LIN {X 0,Y 523.916,Z 118.035,A -85,B 0,C 180,E1 -4641.08,E2 -4641.08} C_VEL
LIN {X 0,Y 523.924,Z 118.033,A -85,B 0,C 180,E1 -4643.827,E2 -4643.827} C_VEL
LIN {X 0,Y 523.941,Z 118.03,A -85,B 0,C 180,E1 -4646.635,E2 -4646.635} C_VEL
LIN {X 0,Y 523.955,Z 118.032,A -85,B 0,C 180,E1 -4649.356,E2 -4649.356} C_VEL
LIN {X 0,Y 523.976,Z 118.024,A -85,B 0,C 180,E1 -4652.281,E2 -4652.281} C_VEL
LIN {X 0,Y 523.951,Z 118.031,A -85,B 0,C 180,E1 -4654.581,E2 -4654.581} C_VEL
LIN {X 0,Y 523.91,Z 118.037,A -85,B 0,C 180,E1 -4657.106,E2 -4657.106} C_VEL
LIN {X 0,Y 523.978,Z 118.024,A -85,B 0,C 180,E1 -4659.866,E2 -4659.866} C_VEL
LIN {X 0,Y 523.966,Z 118.031,A -85,B 0,C 180,E1 -4662.837,E2 -4662.837} C_VEL
LIN {X 0,Y 523.976,Z 118.025,A -85,B 0,C 180,E1 -4665.236,E2 -4665.236} C_VEL
LIN {X 0,Y 524.014,Z 118.028,A -85,B 0,C 180,E1 -4668.394,E2 -4668.394} C_VEL
LIN {X 0,Y 524.002,Z 118.021,A -85,B 0,C 180,E1 -4671.516,E2 -4671.516} C_VEL
LIN {X 0,Y 524.081,Z 118.014,A -85,B 0,C 180,E1 -4674.614,E2 -4674.614} C_VEL
LIN {X 0,Y 524.112,Z 118.011,A -85,B 0,C 180,E1 -4677.694,E2 -4677.694} C_VEL
LIN {X 0,Y 524.122,Z 118.006,A -85,B 0,C 180,E1 -4680.768,E2 -4680.768} C_VEL
LIN {X 0,Y 524.07,Z 118.013,A -85,B 0,C 180,E1 -4683.075,E2 -4683.075} C_VEL
LIN {X 0,Y 524.045,Z 118.018,A -85,B 0,C 180,E1 -4686.159,E2 -4686.159} C_VEL
LIN {X 0,Y 523.996,Z 118.025,A -85,B 0,C 180,E1 -4689.262,E2 -4689.262} C_VEL
LIN {X 0,Y 524.001,Z 118.026,A -85,B 0,C 180,E1 -4691.739,E2 -4691.739} C_VEL
LIN {X 0,Y 523.992,Z 118.026,A -85,B 0,C 180,E1 -4695.052,E2 -4695.052} C_VEL
LIN {X 0,Y 523.963,Z 118.026,A -85,B 0,C 180,E1 -4697.969,E2 -4697.969} C_VEL
LIN {X 0,Y 523.971,Z 118.025,A -85,B 0,C 180,E1 -4700.41,E2 -4700.41} C_VEL
LIN {X 0,Y 523.909,Z 118.038,A -85,B 0,C 180,E1 -4702.894,E2 -4702.894} C_VEL
LIN {X 0,Y 523.95,Z 118.03,A -85,B 0,C 180,E1 -4705.419,E2 -4705.419} C_VEL
LIN {X 0,Y 523.966,Z 118.025,A -85,B 0,C 180,E1 -4707.999,E2 -4707.999} C_VEL
LIN {X 0,Y 523.943,Z 118.036,A -85,B 0,C 180,E1 -4710.855,E2 -4710.855} C_VEL
LIN {X 0,Y 523.959,Z 118.026,A -85,B 0,C 180,E1 -4713.735,E2 -4713.735} C_VEL
LIN {X 0,Y 523.918,Z 118.037,A -85,B 0,C 180,E1 -4716.404,E2 -4716.404} C_VEL
LIN {X 0,Y 523.918,Z 118.032,A -85,B 0,C 180,E1 -4719.085,E2 -4719.085} C_VEL
LIN {X 0,Y 523.952,Z 118.032,A -85,B 0,C 180,E1 -4722.119,E2 -4722.119} C_VEL
LIN {X 0,Y 523.942,Z 118.028,A -85,B 0,C 180,E1 -4725.31,E2 -4725.31} C_VEL
LIN {X 0,Y 523.956,Z 118.028,A -85,B 0,C 180,E1 -4728.69,E2 -4728.69} C_VEL
LIN {X 0,Y 523.915,Z 118.031,A -85,B 0,C 180,E1 -4731.081,E2 -4731.081} C_VEL
LIN {X 0,Y 523.922,Z 118.038,A -85,B 0,C 180,E1 -4733.827,E2 -4733.827} C_VEL
LIN {X 0,Y 523.913,Z 118.032,A -85,B 0,C 180,E1 -4736.634,E2 -4736.634} C_VEL
LIN {X 0,Y 523.955,Z 118.03,A -85,B 0,C 180,E1 -4739.356,E2 -4739.356} C_VEL
LIN {X 0,Y 523.976,Z 118.025,A -85,B 0,C 180,E1 -4742.282,E2 -4742.282} C_VEL
LIN {X 0,Y 523.951,Z 118.028,A -85,B 0,C 180,E1 -4744.582,E2 -4744.582} C_VEL
LIN {X 0,Y 523.909,Z 118.018,A -85,B 0,C 180,E1 -4747.107,E2 -4747.107} C_VEL
LIN {X 0,Y 523.971,Z 118.238,A -85,B 0,C 180,E1 -4748.097,E2 -4748.097} C_VEL
LIN {X 0,Y 524.691,Z 123.717,A -85,B 0,C 180,E1 -4749.21,E2 -4749.21} C_VEL
LIN {X 0,Y 524.349,Z 138.793,A -85,B 0,C 180,E1 -4752.107,E2 -4752.107} C_VEL
LIN {X 0,Y 524.033,Z 153.682,A -85,B 0,C 180,E1 -4754.932,E2 -4754.932} C_VEL
LIN {X 0,Y 523.832,Z 170.237,A -85,B 0,C 180,E1 -4758.019,E2 -4758.019} C_VEL
LIN {X 0,Y 523.848,Z 170.802,A -85,B 0,C 180,E1 -4758.075,E2 -4758.075} C_VEL
LIN {X 0,Y 524.951,Z 180.485,A -85,B 0,C 180,E1 -4758.254,E2 -4758.254} C_VEL
LIN {X 0,Y 524.795,Z 246.49,A -85,B 0,C 180,E1 -4759.17,E2 -4759.17} C_VEL
LIN {X 0,Y 524.624,Z 255.76,A -85,B 0,C 180,E1 -4759.386,E2 -4759.386} C_VEL
LIN {X 0,Y 524.521,Z 264.237,A -85,B 0,C 180,E1 -4759.676,E2 -4759.676} C_VEL
LIN {X 0,Y 524.401,Z 272.75,A -85,B 0,C 180,E1 -4760.064,E2 -4760.064} C_VEL
LIN {X 0,Y 524.221,Z 281.094,A -85,B 0,C 180,E1 -4760.548,E2 -4760.548} C_VEL
LIN {X 0,Y 524.065,Z 289.144,A -85,B 0,C 180,E1 -4761.129,E2 -4761.129} C_VEL
LIN {X 0,Y 523.853,Z 297.832,A -85,B 0,C 180,E1 -4761.902,E2 -4761.902} C_VEL
LIN {X 0,Y 523.702,Z 306.356,A -85,B 0,C 180,E1 -4762.869,E2 -4762.869} C_VEL
LIN {X 0,Y 523.612,Z 313.045,A -85,B 0,C 180,E1 -4763.836,E2 -4763.836} C_VEL
LIN {X 0,Y 523.484,Z 317.435,A -85,B 0,C 180,E1 -4764.608,E2 -4764.608} C_VEL
LIN {X 0,Y 523.465,Z 322.611,A -85,B 0,C 180,E1 -4765.765,E2 -4765.765} C_VEL
LIN {X 0,Y 523.407,Z 325.256,A -85,B 0,C 180,E1 -4766.536,E2 -4766.536} C_VEL
LIN {X 0,Y 523.336,Z 328.158,A -85,B 0,C 180,E1 -4767.691,E2 -4767.691} C_VEL
LIN {X 0,Y 523.273,Z 329.409,A -85,B 0,C 180,E1 -4768.461,E2 -4768.461} C_VEL
LIN {X 0,Y 523.248,Z 330.188,A -85,B 0,C 180,E1 -4769.231,E2 -4769.231} C_VEL
LIN {X 0,Y 523.247,Z 330.484,A -85,B 0,C 180,E1 -4770,E2 -4770} C_VEL
LIN {X 0,Y 523.248,Z 330.188,A -85,B 0,C 180,E1 -4770.77,E2 -4770.77} C_VEL
LIN {X 0,Y 523.273,Z 329.408,A -85,B 0,C 180,E1 -4771.539,E2 -4771.539} C_VEL
LIN {X 0,Y 523.336,Z 328.156,A -85,B 0,C 180,E1 -4772.309,E2 -4772.309} C_VEL
LIN {X 0,Y 523.407,Z 325.254,A -85,B 0,C 180,E1 -4773.464,E2 -4773.464} C_VEL
LIN {X 0,Y 523.465,Z 322.609,A -85,B 0,C 180,E1 -4774.235,E2 -4774.235} C_VEL
LIN {X 0,Y 523.484,Z 317.43,A -85,B 0,C 180,E1 -4775.393,E2 -4775.393} C_VEL
LIN {X 0,Y 523.599,Z 311.458,A -85,B 0,C 180,E1 -4776.424,E2 -4776.424} C_VEL
LIN {X 0,Y 523.697,Z 304.846,A -85,B 0,C 180,E1 -4777.325,E2 -4777.325} C_VEL
LIN {X 0,Y 523.897,Z 296.813,A -85,B 0,C 180,E1 -4778.195,E2 -4778.195} C_VEL
LIN {X 0,Y 524.065,Z 289.143,A -85,B 0,C 180,E1 -4778.872,E2 -4778.872} C_VEL
LIN {X 0,Y 524.24,Z 281.089,A -85,B 0,C 180,E1 -4779.452,E2 -4779.452} C_VEL
LIN {X 0,Y 524.394,Z 272.745,A -85,B 0,C 180,E1 -4779.936,E2 -4779.936} C_VEL
LIN {X 0,Y 524.546,Z 264.232,A -85,B 0,C 180,E1 -4780.323,E2 -4780.323} C_VEL
LIN {X 0,Y 524.635,Z 254.085,A -85,B 0,C 180,E1 -4780.663,E2 -4780.663} C_VEL
LIN {X 0,Y 524.826,Z 242.383,A -85,B 0,C 180,E1 -4780.903,E2 -4780.903} C_VEL
LIN {X 0,Y 524.778,Z 178.186,A -85,B 0,C 180,E1 -4781.782,E2 -4781.782} C_VEL
LIN {X 0,Y 523.851,Z 170.702,A -85,B 0,C 180,E1 -4781.93,E2 -4781.93} C_VEL
LIN {X 0,Y 523.841,Z 164.752,A -85,B 0,C 180,E1 -4782.987,E2 -4782.987} C_VEL
LIN {X 0,Y 524.091,Z 151.089,A -85,B 0,C 180,E1 -4785.557,E2 -4785.557} C_VEL
LIN {X 0,Y 524.457,Z 134.255,A -85,B 0,C 180,E1 -4788.761,E2 -4788.761} C_VEL
LIN {X 0,Y 524.69,Z 122.657,A -85,B 0,C 180,E1 -4790.996,E2 -4790.996} C_VEL
LIN {X 0,Y 523.958,Z 118.102,A -85,B 0,C 180,E1 -4791.956,E2 -4791.956} C_VEL
LIN {X 0,Y 523.929,Z 118.024,A -85,B 0,C 180,E1 -4794.572,E2 -4794.572} C_VEL
LIN {X 0,Y 523.951,Z 118.028,A -85,B 0,C 180,E1 -4797.133,E2 -4797.133} C_VEL
LIN {X 0,Y 523.943,Z 118.03,A -85,B 0,C 180,E1 -4799.756,E2 -4799.756} C_VEL
LIN {X 0,Y 523.934,Z 118.035,A -85,B 0,C 180,E1 -4802.45,E2 -4802.45} C_VEL
LIN {X 0,Y 523.921,Z 118.031,A -85,B 0,C 180,E1 -4805.227,E2 -4805.227} C_VEL
LIN {X 0,Y 523.916,Z 118.039,A -85,B 0,C 180,E1 -4808.102,E2 -4808.102} C_VEL
LIN {X 0,Y 523.939,Z 118.029,A -85,B 0,C 180,E1 -4811.092,E2 -4811.092} C_VEL
LIN {X 0,Y 523.931,Z 118.032,A -85,B 0,C 180,E1 -4814.229,E2 -4814.229} C_VEL
LIN {X 0,Y 523.917,Z 118.031,A -85,B 0,C 180,E1 -4816.833,E2 -4816.833} C_VEL
LIN {X 0,Y 523.941,Z 118.029,A -85,B 0,C 180,E1 -4818.908,E2 -4818.908} C_VEL
LIN {X 0,Y 523.917,Z 118.035,A -85,B 0,C 180,E1 -4821.898,E2 -4821.898} C_VEL
LIN {X 0,Y 523.936,Z 118.031,A -85,B 0,C 180,E1 -4824.91,E2 -4824.91} C_VEL
LIN {X 0,Y 523.936,Z 118.032,A -85,B 0,C 180,E1 -4827.68,E2 -4827.68} C_VEL
LIN {X 0,Y 523.955,Z 118.029,A -85,B 0,C 180,E1 -4830.677,E2 -4830.677} C_VEL
LIN {X 0,Y 523.974,Z 118.025,A -85,B 0,C 180,E1 -4833.729,E2 -4833.729} C_VEL
LIN {X 0,Y 523.926,Z 118.031,A -85,B 0,C 180,E1 -4836.27,E2 -4836.27} C_VEL
LIN {X 0,Y 523.948,Z 118.035,A -85,B 0,C 180,E1 -4838.767,E2 -4838.767} C_VEL
LIN {X 0,Y 523.953,Z 118.03,A -85,B 0,C 180,E1 -4841.221,E2 -4841.221} C_VEL
LIN {X 0,Y 523.938,Z 118.029,A -85,B 0,C 180,E1 -4843.639,E2 -4843.639} C_VEL
LIN {X 0,Y 523.941,Z 118.03,A -85,B 0,C 180,E1 -4846.028,E2 -4846.028} C_VEL
LIN {X 0,Y 524.014,Z 118.026,A -85,B 0,C 180,E1 -4848.394,E2 -4848.394} C_VEL
LIN {X 0,Y 524.005,Z 118.02,A -85,B 0,C 180,E1 -4851.516,E2 -4851.516} C_VEL
LIN {X 0,Y 524.082,Z 118.015,A -85,B 0,C 180,E1 -4854.614,E2 -4854.614} C_VEL
LIN {X 0,Y 524.112,Z 118.01,A -85,B 0,C 180,E1 -4857.695,E2 -4857.695} C_VEL
LIN {X 0,Y 524.125,Z 118.006,A -85,B 0,C 180,E1 -4860.768,E2 -4860.768} C_VEL
LIN {X 0,Y 524.071,Z 118.012,A -85,B 0,C 180,E1 -4863.075,E2 -4863.075} C_VEL
LIN {X 0,Y 524.047,Z 118.019,A -85,B 0,C 180,E1 -4866.159,E2 -4866.159} C_VEL
LIN {X 0,Y 523.998,Z 118.024,A -85,B 0,C 180,E1 -4869.262,E2 -4869.262} C_VEL
LIN {X 0,Y 524.027,Z 118.025,A -85,B 0,C 180,E1 -4871.751,E2 -4871.751} C_VEL
LIN {X 0,Y 523.995,Z 118.024,A -85,B 0,C 180,E1 -4875.052,E2 -4875.052} C_VEL
LIN {X 0,Y 523.965,Z 118.027,A -85,B 0,C 180,E1 -4877.969,E2 -4877.969} C_VEL
LIN {X 0,Y 523.974,Z 118.024,A -85,B 0,C 180,E1 -4880.41,E2 -4880.41} C_VEL
LIN {X 0,Y 523.912,Z 118.036,A -85,B 0,C 180,E1 -4882.894,E2 -4882.894} C_VEL
LIN {X 0,Y 523.986,Z 118.023,A -85,B 0,C 180,E1 -4886.02,E2 -4886.02} C_VEL
LIN {X 0,Y 523.941,Z 118.036,A -85,B 0,C 180,E1 -4888.875,E2 -4888.875} C_VEL
LIN {X 0,Y 523.922,Z 118.032,A -85,B 0,C 180,E1 -4891.544,E2 -4891.544} C_VEL
LIN {X 0,Y 523.943,Z 118.03,A -85,B 0,C 180,E1 -4894.29,E2 -4894.29} C_VEL
LIN {X 0,Y 523.913,Z 118.034,A -85,B 0,C 180,E1 -4897.132,E2 -4897.132} C_VEL
LIN {X 0,Y 523.939,Z 118.031,A -85,B 0,C 180,E1 -4900.13,E2 -4900.13} C_VEL
LIN {X 0,Y 523.936,Z 118.038,A -85,B 0,C 180,E1 -4902.459,E2 -4902.459} C_VEL
LIN {X 0,Y 523.943,Z 118.028,A -85,B 0,C 180,E1 -4905.31,E2 -4905.31} C_VEL
LIN {X 0,Y 523.916,Z 118.033,A -85,B 0,C 180,E1 -4906.907,E2 -4906.907} C_VEL
LIN {X 0,Y 523.252,Z 118.115,A -85,B 0,C 180,E1 -4907.548,E2 -4907.548} C_VEL
LIN {X 0,Y 520.412,Z 118.477,A -85,B 0,C 180,E1 -4908.59,E2 -4908.59} C_VEL
LIN {X 0,Y 518.008,Z 118.781,A -85,B 0,C 180,E1 -4909.429,E2 -4909.429} C_VEL
LIN {X 0,Y 516.97,Z 118.907,A -85,B 0,C 180,E1 -4910.077,E2 -4910.077} C_VEL
LIN {X 0,Y 516.883,Z 118.915,A -85,B 0,C 180,E1 -4910.296,E2 -4910.296} C_VEL
LIN {X 0,Y 516.886,Z 118.908,A -85,B 0,C 180,E1 -4913.342,E2 -4913.342} C_VEL
LIN {X 0,Y 516.891,Z 118.913,A -85,B 0,C 180,E1 -4916.119,E2 -4916.119} C_VEL
LIN {X 0,Y 516.893,Z 118.906,A -85,B 0,C 180,E1 -4918.936,E2 -4918.936} C_VEL
LIN {X 0,Y 516.92,Z 118.909,A -85,B 0,C 180,E1 -4921.585,E2 -4921.585} C_VEL
LIN {X 0,Y 516.932,Z 118.903,A -85,B 0,C 180,E1 -4924.211,E2 -4924.211} C_VEL
LIN {X 0,Y 516.862,Z 118.912,A -85,B 0,C 180,E1 -4926.776,E2 -4926.776} C_VEL
LIN {X 0,Y 516.942,Z 118.908,A -85,B 0,C 180,E1 -4929.732,E2 -4929.732} C_VEL
LIN {X 0,Y 516.999,Z 119.097,A -85,B 0,C 180,E1 -4930.598,E2 -4930.598} C_VEL
LIN {X 0,Y 517.204,Z 126.654,A -85,B 0,C 180,E1 -4932.306,E2 -4932.306} C_VEL
LIN {X 0,Y 516.92,Z 140.888,A -85,B 0,C 180,E1 -4935.432,E2 -4935.432} C_VEL
LIN {X 0,Y 516.764,Z 152.656,A -85,B 0,C 180,E1 -4937.928,E2 -4937.928} C_VEL
LIN {X 0,Y 516.959,Z 154.363,A -85,B 0,C 180,E1 -4938.008,E2 -4938.008} C_VEL
LIN {X 0,Y 518.088,Z 162.675,A -85,B 0,C 180,E1 -4938.15,E2 -4938.15} C_VEL
LIN {X 0,Y 517.826,Z 228.184,A -85,B 0,C 180,E1 -4939.071,E2 -4939.071} C_VEL
LIN {X 0,Y 517.719,Z 237.369,A -85,B 0,C 180,E1 -4939.292,E2 -4939.292} C_VEL
LIN {X 0,Y 517.622,Z 247.003,A -85,B 0,C 180,E1 -4939.636,E2 -4939.636} C_VEL
LIN {X 0,Y 517.469,Z 255.2,A -85,B 0,C 180,E1 -4940.028,E2 -4940.028} C_VEL
LIN {X 0,Y 517.248,Z 264.818,A -85,B 0,C 180,E1 -4940.616,E2 -4940.616} C_VEL
LIN {X 0,Y 517.002,Z 274.654,A -85,B 0,C 180,E1 -4941.4,E2 -4941.4} C_VEL
LIN {X 0,Y 516.806,Z 282.4,A -85,B 0,C 180,E1 -4942.184,E2 -4942.184} C_VEL
LIN {X 0,Y 516.668,Z 288.767,A -85,B 0,C 180,E1 -4942.968,E2 -4942.968} C_VEL
LIN {X 0,Y 516.654,Z 294.059,A -85,B 0,C 180,E1 -4943.752,E2 -4943.752} C_VEL
LIN {X 0,Y 516.435,Z 298.481,A -85,B 0,C 180,E1 -4944.533,E2 -4944.533} C_VEL
LIN {X 0,Y 516.425,Z 303.674,A -85,B 0,C 180,E1 -4945.707,E2 -4945.707} C_VEL
LIN {X 0,Y 516.354,Z 306.346,A -85,B 0,C 180,E1 -4946.488,E2 -4946.488} C_VEL
LIN {X 0,Y 516.266,Z 309.27,A -85,B 0,C 180,E1 -4947.659,E2 -4947.659} C_VEL
LIN {X 0,Y 516.191,Z 310.553,A -85,B 0,C 180,E1 -4948.439,E2 -4948.439} C_VEL
LIN {X 0,Y 516.159,Z 311.366,A -85,B 0,C 180,E1 -4949.22,E2 -4949.22} C_VEL
LIN {X 0,Y 516.155,Z 311.675,A -85,B 0,C 180,E1 -4950,E2 -4950} C_VEL
LIN {X 0,Y 516.16,Z 311.403,A -85,B 0,C 180,E1 -4950.78,E2 -4950.78} C_VEL
LIN {X 0,Y 516.192,Z 310.665,A -85,B 0,C 180,E1 -4951.56,E2 -4951.56} C_VEL
LIN {X 0,Y 516.266,Z 309.457,A -85,B 0,C 180,E1 -4952.34,E2 -4952.34} C_VEL
LIN {X 0,Y 516.342,Z 306.612,A -85,B 0,C 180,E1 -4953.511,E2 -4953.511} C_VEL
LIN {X 0,Y 516.421,Z 304.024,A -85,B 0,C 180,E1 -4954.292,E2 -4954.292} C_VEL
LIN {X 0,Y 516.431,Z 298.924,A -85,B 0,C 180,E1 -4955.466,E2 -4955.466} C_VEL
LIN {X 0,Y 516.674,Z 292.958,A -85,B 0,C 180,E1 -4956.523,E2 -4956.523} C_VEL
LIN {X 0,Y 516.761,Z 284.877,A -85,B 0,C 180,E1 -4957.62,E2 -4957.62} C_VEL
LIN {X 0,Y 516.949,Z 277.621,A -85,B 0,C 180,E1 -4958.404,E2 -4958.404} C_VEL
LIN {X 0,Y 517.168,Z 269.868,A -85,B 0,C 180,E1 -4959.089,E2 -4959.089} C_VEL
LIN {X 0,Y 517.291,Z 261.695,A -85,B 0,C 180,E1 -4959.679,E2 -4959.679} C_VEL
LIN {X 0,Y 517.509,Z 253.168,A -85,B 0,C 180,E1 -4960.168,E2 -4960.168} C_VEL
LIN {X 0,Y 517.647,Z 243.167,A -85,B 0,C 180,E1 -4960.611,E2 -4960.611} C_VEL
LIN {X 0,Y 517.888,Z 231.618,A -85,B 0,C 180,E1 -4960.952,E2 -4960.952} C_VEL
LIN {X 0,Y 517.888,Z 214.705,A -85,B 0,C 180,E1 -4961.223,E2 -4961.223} C_VEL
LIN {X 0,Y 517.941,Z 160.898,A -85,B 0,C 180,E1 -4961.968,E2 -4961.968} C_VEL
LIN {X 0,Y 516.808,Z 153.119,A -85,B 0,C 180,E1 -4962.124,E2 -4962.124} C_VEL
LIN {X 0,Y 516.767,Z 152.014,A -85,B 0,C 180,E1 -4962.269,E2 -4962.269} C_VEL
LIN {X 0,Y 516.971,Z 137.489,A -85,B 0,C 180,E1 -4965.398,E2 -4965.398} C_VEL
LIN {X 0,Y 517.247,Z 124.737,A -85,B 0,C 180,E1 -4968.21,E2 -4968.21} C_VEL
LIN {X 0,Y 517.004,Z 118.99,A -85,B 0,C 180,E1 -4969.557,E2 -4969.557} C_VEL
LIN {X 0,Y 516.867,Z 118.917,A -85,B 0,C 180,E1 -4972.389,E2 -4972.389} C_VEL
LIN {X 0,Y 516.875,Z 118.911,A -85,B 0,C 180,E1 -4974.93,E2 -4974.93} C_VEL
LIN {X 0,Y 516.927,Z 118.902,A -85,B 0,C 180,E1 -4977.532,E2 -4977.532} C_VEL
LIN {X 0,Y 516.892,Z 118.914,A -85,B 0,C 180,E1 -4980.203,E2 -4980.203} C_VEL
LIN {X 0,Y 516.882,Z 118.908,A -85,B 0,C 180,E1 -4982.948,E2 -4982.948} C_VEL
LIN {X 0,Y 516.887,Z 118.912,A -85,B 0,C 180,E1 -4985.779,E2 -4985.779} C_VEL
LIN {X 0,Y 516.88,Z 118.908,A -85,B 0,C 180,E1 -4988.716,E2 -4988.716} C_VEL
LIN {X 0,Y 516.911,Z 118.912,A -85,B 0,C 180,E1 -4991.775,E2 -4991.775} C_VEL
LIN {X 0,Y 516.894,Z 118.907,A -85,B 0,C 180,E1 -4995.007,E2 -4995.007} C_VEL
LIN {X 0,Y 516.914,Z 118.904,A -85,B 0,C 180,E1 -4998.398,E2 -4998.398} C_VEL
LIN {X 0,Y 516.88,Z 118.914,A -85,B 0,C 180,E1 -5001.284,E2 -5001.284} C_VEL
LIN {X 0,Y 516.887,Z 118.907,A -85,B 0,C 180,E1 -5004.221,E2 -5004.221} C_VEL
LIN {X 0,Y 516.894,Z 118.912,A -85,B 0,C 180,E1 -5007.053,E2 -5007.053} C_VEL
LIN {X 0,Y 516.891,Z 118.908,A -85,B 0,C 180,E1 -5009.796,E2 -5009.796} C_VEL
LIN {X 0,Y 516.925,Z 118.904,A -85,B 0,C 180,E1 -5012.467,E2 -5012.467} C_VEL
LIN {X 0,Y 516.908,Z 118.911,A -85,B 0,C 180,E1 -5015.072,E2 -5015.072} C_VEL
LIN {X 0,Y 516.885,Z 118.911,A -85,B 0,C 180,E1 -5018.462,E2 -5018.462} C_VEL
LIN {X 0,Y 516.903,Z 118.91,A -85,B 0,C 180,E1 -5020.955,E2 -5020.955} C_VEL
LIN {X 0,Y 516.913,Z 118.904,A -85,B 0,C 180,E1 -5023.41,E2 -5023.41} C_VEL
LIN {X 0,Y 516.894,Z 118.907,A -85,B 0,C 180,E1 -5025.834,E2 -5025.834} C_VEL
LIN {X 0,Y 517.004,Z 118.898,A -85,B 0,C 180,E1 -5028.234,E2 -5028.234} C_VEL
LIN {X 0,Y 516.967,Z 118.897,A -85,B 0,C 180,E1 -5031.4,E2 -5031.4} C_VEL
LIN {X 0,Y 517.01,Z 118.894,A -85,B 0,C 180,E1 -5033.757,E2 -5033.757} C_VEL
LIN {X 0,Y 517.084,Z 118.886,A -85,B 0,C 180,E1 -5037.663,E2 -5037.663} C_VEL
LIN {X 0,Y 517.092,Z 118.882,A -85,B 0,C 180,E1 -5040.779,E2 -5040.779} C_VEL
LIN {X 0,Y 517.011,Z 118.892,A -85,B 0,C 180,E1 -5043.117,E2 -5043.117} C_VEL
LIN {X 0,Y 517.009,Z 118.894,A -85,B 0,C 180,E1 -5046.243,E2 -5046.243} C_VEL
LIN {X 0,Y 516.95,Z 118.905,A -85,B 0,C 180,E1 -5049.389,E2 -5049.389} C_VEL
LIN {X 0,Y 516.951,Z 118.904,A -85,B 0,C 180,E1 -5051.807,E2 -5051.807} C_VEL
LIN {X 0,Y 516.943,Z 118.905,A -85,B 0,C 180,E1 -5055.146,E2 -5055.146} C_VEL
LIN {X 0,Y 516.924,Z 118.902,A -85,B 0,C 180,E1 -5058.222,E2 -5058.222} C_VEL
LIN {X 0,Y 516.911,Z 118.906,A -85,B 0,C 180,E1 -5060.701,E2 -5060.701} C_VEL
LIN {X 0,Y 516.901,Z 118.905,A -85,B 0,C 180,E1 -5064.072,E2 -5064.072} C_VEL
LIN {X 0,Y 516.923,Z 118.907,A -85,B 0,C 180,E1 -5066.658,E2 -5066.658} C_VEL
LIN {X 0,Y 516.909,Z 118.905,A -85,B 0,C 180,E1 -5069.524,E2 -5069.524} C_VEL
LIN {X 0,Y 516.894,Z 118.912,A -85,B 0,C 180,E1 -5072.543,E2 -5072.543} C_VEL
LIN {X 0,Y 516.878,Z 118.909,A -85,B 0,C 180,E1 -5075.332,E2 -5075.332} C_VEL
LIN {X 0,Y 516.879,Z 118.91,A -85,B 0,C 180,E1 -5077.943,E2 -5077.943} C_VEL
LIN {X 0,Y 516.882,Z 118.912,A -85,B 0,C 180,E1 -5080.742,E2 -5080.742} C_VEL
LIN {X 0,Y 516.882,Z 118.91,A -85,B 0,C 180,E1 -5082.831,E2 -5082.831} C_VEL
LIN {X 0,Y 516.893,Z 118.907,A -85,B 0,C 180,E1 -5085.007,E2 -5085.007} C_VEL
LIN {X 0,Y 516.913,Z 118.908,A -85,B 0,C 180,E1 -5088.399,E2 -5088.399} C_VEL
LIN {X 0,Y 516.879,Z 118.909,A -85,B 0,C 180,E1 -5091.284,E2 -5091.284} C_VEL
LIN {X 0,Y 516.886,Z 118.911,A -85,B 0,C 180,E1 -5094.221,E2 -5094.221} C_VEL
LIN {X 0,Y 516.88,Z 118.908,A -85,B 0,C 180,E1 -5097.052,E2 -5097.052} C_VEL
LIN {X 0,Y 516.891,Z 118.914,A -85,B 0,C 180,E1 -5099.797,E2 -5099.797} C_VEL
LIN {X 0,Y 516.925,Z 118.902,A -85,B 0,C 180,E1 -5102.468,E2 -5102.468} C_VEL
LIN {X 0,Y 516.907,Z 118.907,A -85,B 0,C 180,E1 -5105.072,E2 -5105.072} C_VEL
LIN {X 0,Y 516.941,Z 119.002,A -85,B 0,C 180,E1 -5107.941,E2 -5107.941} C_VEL
LIN {X 0,Y 517.708,Z 124.653,A -85,B 0,C 180,E1 -5109.124,E2 -5109.124} C_VEL
LIN {X 0,Y 517.336,Z 139.312,A -85,B 0,C 180,E1 -5111.98,E2 -5111.98} C_VEL
LIN {X 0,Y 516.992,Z 154.151,A -85,B 0,C 180,E1 -5114.835,E2 -5114.835} C_VEL
LIN {X 0,Y 516.784,Z 169.971,A -85,B 0,C 180,E1 -5117.831,E2 -5117.831} C_VEL
LIN {X 0,Y 516.82,Z 170.959,A -85,B 0,C 180,E1 -5117.922,E2 -5117.922} C_VEL
LIN {X 0,Y 517.994,Z 181.342,A -85,B 0,C 180,E1 -5118.107,E2 -5118.107} C_VEL
LIN {X 0,Y 517.832,Z 246.386,A -85,B 0,C 180,E1 -5119.023,E2 -5119.023} C_VEL
LIN {X 0,Y 517.657,Z 255.631,A -85,B 0,C 180,E1 -5119.241,E2 -5119.241} C_VEL
LIN {X 0,Y 517.548,Z 264.109,A -85,B 0,C 180,E1 -5119.536,E2 -5119.536} C_VEL
LIN {X 0,Y 517.402,Z 272.622,A -85,B 0,C 180,E1 -5119.928,E2 -5119.928} C_VEL
LIN {X 0,Y 517.198,Z 280.965,A -85,B 0,C 180,E1 -5120.418,E2 -5120.418} C_VEL
LIN {X 0,Y 517.043,Z 289.015,A -85,B 0,C 180,E1 -5121.007,E2 -5121.007} C_VEL
LIN {X 0,Y 516.811,Z 297.703,A -85,B 0,C 180,E1 -5121.791,E2 -5121.791} C_VEL
LIN {X 0,Y 516.649,Z 306.228,A -85,B 0,C 180,E1 -5122.772,E2 -5122.772} C_VEL
LIN {X 0,Y 516.521,Z 312.916,A -85,B 0,C 180,E1 -5123.751,E2 -5123.751} C_VEL
LIN {X 0,Y 516.43,Z 317.307,A -85,B 0,C 180,E1 -5124.534,E2 -5124.534} C_VEL
LIN {X 0,Y 516.368,Z 322.483,A -85,B 0,C 180,E1 -5125.707,E2 -5125.707} C_VEL
LIN {X 0,Y 516.324,Z 325.128,A -85,B 0,C 180,E1 -5126.489,E2 -5126.489} C_VEL
LIN {X 0,Y 516.262,Z 328.029,A -85,B 0,C 180,E1 -5127.66,E2 -5127.66} C_VEL
LIN {X 0,Y 516.19,Z 329.281,A -85,B 0,C 180,E1 -5128.44,E2 -5128.44} C_VEL
LIN {X 0,Y 516.158,Z 330.06,A -85,B 0,C 180,E1 -5129.22,E2 -5129.22} C_VEL
LIN {X 0,Y 516.154,Z 330.355,A -85,B 0,C 180,E1 -5130,E2 -5130} C_VEL
LIN {X 0,Y 516.158,Z 330.06,A -85,B 0,C 180,E1 -5130.78,E2 -5130.78} C_VEL
LIN {X 0,Y 516.19,Z 329.279,A -85,B 0,C 180,E1 -5131.561,E2 -5131.561} C_VEL
LIN {X 0,Y 516.262,Z 328.028,A -85,B 0,C 180,E1 -5132.341,E2 -5132.341} C_VEL
LIN {X 0,Y 516.324,Z 325.126,A -85,B 0,C 180,E1 -5133.512,E2 -5133.512} C_VEL
LIN {X 0,Y 516.368,Z 322.481,A -85,B 0,C 180,E1 -5134.293,E2 -5134.293} C_VEL
LIN {X 0,Y 516.43,Z 317.302,A -85,B 0,C 180,E1 -5135.467,E2 -5135.467} C_VEL
LIN {X 0,Y 516.507,Z 311.945,A -85,B 0,C 180,E1 -5136.41,E2 -5136.41} C_VEL
LIN {X 0,Y 516.627,Z 304.717,A -85,B 0,C 180,E1 -5137.426,E2 -5137.426} C_VEL
LIN {X 0,Y 516.847,Z 296.684,A -85,B 0,C 180,E1 -5138.307,E2 -5138.307} C_VEL
LIN {X 0,Y 517.043,Z 289.015,A -85,B 0,C 180,E1 -5138.993,E2 -5138.993} C_VEL
LIN {X 0,Y 517.231,Z 280.961,A -85,B 0,C 180,E1 -5139.582,E2 -5139.582} C_VEL
LIN {X 0,Y 517.397,Z 272.617,A -85,B 0,C 180,E1 -5140.072,E2 -5140.072} C_VEL
LIN {X 0,Y 517.535,Z 264.103,A -85,B 0,C 180,E1 -5140.465,E2 -5140.465} C_VEL
LIN {X 0,Y 517.665,Z 253.957,A -85,B 0,C 180,E1 -5140.808,E2 -5140.808} C_VEL
LIN {X 0,Y 517.878,Z 242.439,A -85,B 0,C 180,E1 -5141.049,E2 -5141.049} C_VEL
LIN {X 0,Y 517.871,Z 179.197,A -85,B 0,C 180,E1 -5141.925,E2 -5141.925} C_VEL
LIN {X 0,Y 516.773,Z 170.582,A -85,B 0,C 180,E1 -5142.096,E2 -5142.096} C_VEL
LIN {X 0,Y 516.785,Z 165.68,A -85,B 0,C 180,E1 -5142.967,E2 -5142.967} C_VEL
LIN {X 0,Y 517.048,Z 152.891,A -85,B 0,C 180,E1 -5145.406,E2 -5145.406} C_VEL
LIN {X 0,Y 517.425,Z 136.242,A -85,B 0,C 180,E1 -5148.614,E2 -5148.614} C_VEL
LIN {X 0,Y 517.694,Z 123.59,A -85,B 0,C 180,E1 -5151.085,E2 -5151.085} C_VEL
LIN {X 0,Y 516.93,Z 118.946,A -85,B 0,C 180,E1 -5152.087,E2 -5152.087} C_VEL
LIN {X 0,Y 516.906,Z 118.907,A -85,B 0,C 180,E1 -5154.928,E2 -5154.928} C_VEL
LIN {X 0,Y 516.926,Z 118.904,A -85,B 0,C 180,E1 -5157.905,E2 -5157.905} C_VEL
LIN {X 0,Y 516.893,Z 118.913,A -85,B 0,C 180,E1 -5160.204,E2 -5160.204} C_VEL
LIN {X 0,Y 516.895,Z 118.907,A -85,B 0,C 180,E1 -5162.947,E2 -5162.947} C_VEL
LIN {X 0,Y 516.872,Z 118.913,A -85,B 0,C 180,E1 -5165.78,E2 -5165.78} C_VEL
LIN {X 0,Y 516.881,Z 118.908,A -85,B 0,C 180,E1 -5168.716,E2 -5168.716} C_VEL
LIN {X 0,Y 516.912,Z 118.911,A -85,B 0,C 180,E1 -5171.775,E2 -5171.775} C_VEL
LIN {X 0,Y 516.895,Z 118.906,A -85,B 0,C 180,E1 -5175.007,E2 -5175.007} C_VEL
LIN {X 0,Y 516.916,Z 118.904,A -85,B 0,C 180,E1 -5178.399,E2 -5178.399} C_VEL
LIN {X 0,Y 516.881,Z 118.913,A -85,B 0,C 180,E1 -5181.284,E2 -5181.284} C_VEL
LIN {X 0,Y 516.889,Z 118.907,A -85,B 0,C 180,E1 -5184.221,E2 -5184.221} C_VEL
LIN {X 0,Y 516.896,Z 118.911,A -85,B 0,C 180,E1 -5187.053,E2 -5187.053} C_VEL
LIN {X 0,Y 516.893,Z 118.908,A -85,B 0,C 180,E1 -5189.796,E2 -5189.796} C_VEL
LIN {X 0,Y 516.927,Z 118.903,A -85,B 0,C 180,E1 -5192.467,E2 -5192.467} C_VEL
LIN {X 0,Y 516.909,Z 118.912,A -85,B 0,C 180,E1 -5195.072,E2 -5195.072} C_VEL
LIN {X 0,Y 516.887,Z 118.91,A -85,B 0,C 180,E1 -5198.462,E2 -5198.462} C_VEL
LIN {X 0,Y 516.905,Z 118.911,A -85,B 0,C 180,E1 -5200.955,E2 -5200.955} C_VEL
LIN {X 0,Y 516.915,Z 118.904,A -85,B 0,C 180,E1 -5203.41,E2 -5203.41} C_VEL
LIN {X 0,Y 516.896,Z 118.906,A -85,B 0,C 180,E1 -5205.834,E2 -5205.834} C_VEL
LIN {X 0,Y 516.967,Z 118.902,A -85,B 0,C 180,E1 -5208.234,E2 -5208.234} C_VEL
LIN {X 0,Y 516.969,Z 118.897,A -85,B 0,C 180,E1 -5211.4,E2 -5211.4} C_VEL
LIN {X 0,Y 517.011,Z 118.893,A -85,B 0,C 180,E1 -5213.757,E2 -5213.757} C_VEL
LIN {X 0,Y 517.085,Z 118.885,A -85,B 0,C 180,E1 -5217.663,E2 -5217.663} C_VEL
LIN {X 0,Y 517.095,Z 118.882,A -85,B 0,C 180,E1 -5220.779,E2 -5220.779} C_VEL
LIN {X 0,Y 517.012,Z 118.892,A -85,B 0,C 180,E1 -5223.117,E2 -5223.117} C_VEL
LIN {X 0,Y 517.012,Z 118.895,A -85,B 0,C 180,E1 -5226.243,E2 -5226.243} C_VEL
LIN {X 0,Y 516.953,Z 118.903,A -85,B 0,C 180,E1 -5229.389,E2 -5229.389} C_VEL
LIN {X 0,Y 516.986,Z 118.901,A -85,B 0,C 180,E1 -5231.824,E2 -5231.824} C_VEL
LIN {X 0,Y 516.946,Z 118.903,A -85,B 0,C 180,E1 -5235.147,E2 -5235.147} C_VEL
LIN {X 0,Y 516.926,Z 118.902,A -85,B 0,C 180,E1 -5238.222,E2 -5238.222} C_VEL
LIN {X 0,Y 516.914,Z 118.905,A -85,B 0,C 180,E1 -5240.702,E2 -5240.702} C_VEL
LIN {X 0,Y 516.892,Z 118.906,A -85,B 0,C 180,E1 -5244.073,E2 -5244.073} C_VEL
LIN {X 0,Y 516.926,Z 118.905,A -85,B 0,C 180,E1 -5246.658,E2 -5246.658} C_VEL
LIN {X 0,Y 516.913,Z 118.905,A -85,B 0,C 180,E1 -5249.524,E2 -5249.524} C_VEL
LIN {X 0,Y 516.897,Z 118.91,A -85,B 0,C 180,E1 -5252.543,E2 -5252.543} C_VEL
LIN {X 0,Y 516.881,Z 118.909,A -85,B 0,C 180,E1 -5255.332,E2 -5255.332} C_VEL
LIN {X 0,Y 516.882,Z 118.908,A -85,B 0,C 180,E1 -5257.943,E2 -5257.943} C_VEL
LIN {X 0,Y 516.884,Z 118.913,A -85,B 0,C 180,E1 -5260.742,E2 -5260.742} C_VEL
LIN {X 0,Y 516.884,Z 118.911,A -85,B 0,C 180,E1 -5262.832,E2 -5262.832} C_VEL
LIN {X 0,Y 516.896,Z 118.907,A -85,B 0,C 180,E1 -5265.007,E2 -5265.007} C_VEL
LIN {X 0,Y 516.915,Z 118.91,A -85,B 0,C 180,E1 -5268.399,E2 -5268.399} C_VEL
LIN {X 0,Y 516.883,Z 118.915,A -85,B 0,C 180,E1 -5270.296,E2 -5270.296} C_VEL
LIN {X 0,Y 516.212,Z 118.993,A -85,B 0,C 180,E1 -5270.946,E2 -5270.946} C_VEL
LIN {X 0,Y 513.367,Z 119.353,A -85,B 0,C 180,E1 -5272.002,E2 -5272.002} C_VEL
LIN {X 0,Y 510.961,Z 119.652,A -85,B 0,C 180,E1 -5272.852,E2 -5272.852} C_VEL
LIN {X 0,Y 509.92,Z 119.779,A -85,B 0,C 180,E1 -5273.508,E2 -5273.508} C_VEL
LIN {X 0,Y 509.832,Z 119.789,A -85,B 0,C 180,E1 -5273.731,E2 -5273.731} C_VEL
LIN {X 0,Y 509.846,Z 119.786,A -85,B 0,C 180,E1 -5276.538,E2 -5276.538} C_VEL
LIN {X 0,Y 509.847,Z 119.786,A -85,B 0,C 180,E1 -5279.334,E2 -5279.334} C_VEL
LIN {X 0,Y 509.894,Z 119.782,A -85,B 0,C 180,E1 -5282.054,E2 -5282.054} C_VEL
LIN {X 0,Y 509.842,Z 119.785,A -85,B 0,C 180,E1 -5284.702,E2 -5284.702} C_VEL
LIN {X 0,Y 509.828,Z 119.794,A -85,B 0,C 180,E1 -5287.458,E2 -5287.458} C_VEL
LIN {X 0,Y 509.965,Z 119.931,A -85,B 0,C 180,E1 -5290.502,E2 -5290.502} C_VEL
LIN {X 0,Y 510.217,Z 126.969,A -85,B 0,C 180,E1 -5292.121,E2 -5292.121} C_VEL
LIN {X 0,Y 509.892,Z 140.945,A -85,B 0,C 180,E1 -5295.227,E2 -5295.227} C_VEL
LIN {X 0,Y 509.701,Z 152.758,A -85,B 0,C 180,E1 -5297.758,E2 -5297.758} C_VEL
LIN {X 0,Y 509.926,Z 154.426,A -85,B 0,C 180,E1 -5297.838,E2 -5297.838} C_VEL
LIN {X 0,Y 511.15,Z 163.146,A -85,B 0,C 180,E1 -5297.991,E2 -5297.991} C_VEL
LIN {X 0,Y 510.882,Z 228.344,A -85,B 0,C 180,E1 -5298.921,E2 -5298.921} C_VEL
LIN {X 0,Y 510.765,Z 237.517,A -85,B 0,C 180,E1 -5299.144,E2 -5299.144} C_VEL
LIN {X 0,Y 510.64,Z 247.146,A -85,B 0,C 180,E1 -5299.492,E2 -5299.492} C_VEL
LIN {X 0,Y 510.493,Z 255.34,A -85,B 0,C 180,E1 -5299.89,E2 -5299.89} C_VEL
LIN {X 0,Y 510.247,Z 264.956,A -85,B 0,C 180,E1 -5300.486,E2 -5300.486} C_VEL
LIN {X 0,Y 509.989,Z 274.789,A -85,B 0,C 180,E1 -5301.281,E2 -5301.281} C_VEL
LIN {X 0,Y 509.763,Z 282.534,A -85,B 0,C 180,E1 -5302.075,E2 -5302.075} C_VEL
LIN {X 0,Y 509.616,Z 288.9,A -85,B 0,C 180,E1 -5302.87,E2 -5302.87} C_VEL
LIN {X 0,Y 509.585,Z 295.36,A -85,B 0,C 180,E1 -5303.864,E2 -5303.864} C_VEL
LIN {X 0,Y 509.294,Z 300.52,A -85,B 0,C 180,E1 -5304.854,E2 -5304.854} C_VEL
LIN {X 0,Y 509.327,Z 305.295,A -85,B 0,C 180,E1 -5306.044,E2 -5306.044} C_VEL
LIN {X 0,Y 509.239,Z 307.623,A -85,B 0,C 180,E1 -5306.835,E2 -5306.835} C_VEL
LIN {X 0,Y 509.196,Z 309.399,A -85,B 0,C 180,E1 -5307.627,E2 -5307.627} C_VEL
LIN {X 0,Y 509.112,Z 310.682,A -85,B 0,C 180,E1 -5308.418,E2 -5308.418} C_VEL
LIN {X 0,Y 509.072,Z 311.495,A -85,B 0,C 180,E1 -5309.209,E2 -5309.209} C_VEL
LIN {X 0,Y 509.067,Z 311.804,A -85,B 0,C 180,E1 -5310,E2 -5310} C_VEL
LIN {X 0,Y 509.073,Z 311.531,A -85,B 0,C 180,E1 -5310.791,E2 -5310.791} C_VEL
LIN {X 0,Y 509.113,Z 310.792,A -85,B 0,C 180,E1 -5311.582,E2 -5311.582} C_VEL
LIN {X 0,Y 509.195,Z 309.584,A -85,B 0,C 180,E1 -5312.373,E2 -5312.373} C_VEL
LIN {X 0,Y 509.262,Z 306.739,A -85,B 0,C 180,E1 -5313.56,E2 -5313.56} C_VEL
LIN {X 0,Y 509.349,Z 304.15,A -85,B 0,C 180,E1 -5314.352,E2 -5314.352} C_VEL
LIN {X 0,Y 509.382,Z 299.049,A -85,B 0,C 180,E1 -5315.542,E2 -5315.542} C_VEL
LIN {X 0,Y 509.621,Z 293.497,A -85,B 0,C 180,E1 -5316.543,E2 -5316.543} C_VEL
LIN {X 0,Y 509.654,Z 286.673,A -85,B 0,C 180,E1 -5317.527,E2 -5317.527} C_VEL
LIN {X 0,Y 509.92,Z 277.743,A -85,B 0,C 180,E1 -5318.52,E2 -5318.52} C_VEL
LIN {X 0,Y 510.157,Z 269.989,A -85,B 0,C 180,E1 -5319.215,E2 -5319.215} C_VEL
LIN {X 0,Y 510.271,Z 263.313,A -85,B 0,C 180,E1 -5319.713,E2 -5319.713} C_VEL
LIN {X 0,Y 510.487,Z 255.156,A -85,B 0,C 180,E1 -5320.21,E2 -5320.21} C_VEL
LIN {X 0,Y 510.615,Z 246.906,A -85,B 0,C 180,E1 -5320.608,E2 -5320.608} C_VEL
LIN {X 0,Y 510.837,Z 238.015,A -85,B 0,C 180,E1 -5320.929,E2 -5320.929} C_VEL
LIN {X 0,Y 510.944,Z 229.25,A -85,B 0,C 180,E1 -5321.15,E2 -5321.15} C_VEL
LIN {X 0,Y 511.057,Z 161.896,A -85,B 0,C 180,E1 -5322.119,E2 -5322.119} C_VEL
LIN {X 0,Y 509.776,Z 153.339,A -85,B 0,C 180,E1 -5322.285,E2 -5322.285} C_VEL
LIN {X 0,Y 509.724,Z 152.108,A -85,B 0,C 180,E1 -5322.441,E2 -5322.441} C_VEL
LIN {X 0,Y 509.953,Z 137.833,A -85,B 0,C 180,E1 -5325.548,E2 -5325.548} C_VEL
LIN {X 0,Y 510.217,Z 124.754,A -85,B 0,C 180,E1 -5328.47,E2 -5328.47} C_VEL
LIN {X 0,Y 509.952,Z 119.876,A -85,B 0,C 180,E1 -5329.629,E2 -5329.629} C_VEL
LIN {X 0,Y 509.821,Z 119.793,A -85,B 0,C 180,E1 -5332.705,E2 -5332.705} C_VEL
LIN {X 0,Y 509.841,Z 119.785,A -85,B 0,C 180,E1 -5335.298,E2 -5335.298} C_VEL
LIN {X 0,Y 509.897,Z 119.783,A -85,B 0,C 180,E1 -5338.1,E2 -5338.1} C_VEL
LIN {X 0,Y 509.846,Z 119.784,A -85,B 0,C 180,E1 -5341.28,E2 -5341.28} C_VEL
LIN {X 0,Y 509.847,Z 119.791,A -85,B 0,C 180,E1 -5344.201,E2 -5344.201} C_VEL
LIN {X 0,Y 509.818,Z 119.789,A -85,B 0,C 180,E1 -5347.34,E2 -5347.34} C_VEL
LIN {X 0,Y 509.837,Z 119.787,A -85,B 0,C 180,E1 -5350.382,E2 -5350.382} C_VEL
LIN {X 0,Y 509.823,Z 119.788,A -85,B 0,C 180,E1 -5353.062,E2 -5353.062} C_VEL
LIN {X 0,Y 509.822,Z 119.794,A -85,B 0,C 180,E1 -5355.793,E2 -5355.793} C_VEL
LIN {X 0,Y 509.856,Z 119.783,A -85,B 0,C 180,E1 -5358.574,E2 -5358.574} C_VEL
LIN {X 0,Y 509.85,Z 119.787,A -85,B 0,C 180,E1 -5361.786,E2 -5361.786} C_VEL
LIN {X 0,Y 509.842,Z 119.785,A -85,B 0,C 180,E1 -5364.623,E2 -5364.623} C_VEL
LIN {X 0,Y 509.86,Z 119.787,A -85,B 0,C 180,E1 -5367.481,E2 -5367.481} C_VEL
LIN {X 0,Y 509.857,Z 119.783,A -85,B 0,C 180,E1 -5370.273,E2 -5370.273} C_VEL
LIN {X 0,Y 509.883,Z 119.787,A -85,B 0,C 180,E1 -5372.944,E2 -5372.944} C_VEL
LIN {X 0,Y 509.863,Z 119.783,A -85,B 0,C 180,E1 -5375.574,E2 -5375.574} C_VEL
LIN {X 0,Y 509.849,Z 119.789,A -85,B 0,C 180,E1 -5378.998,E2 -5378.998} C_VEL
LIN {X 0,Y 509.888,Z 119.78,A -85,B 0,C 180,E1 -5381.999,E2 -5381.999} C_VEL
LIN {X 0,Y 509.909,Z 119.781,A -85,B 0,C 180,E1 -5384.819,E2 -5384.819} C_VEL
LIN {X 0,Y 509.943,Z 119.776,A -85,B 0,C 180,E1 -5388.101,E2 -5388.101} C_VEL
LIN {X 0,Y 509.914,Z 119.776,A -85,B 0,C 180,E1 -5391.28,E2 -5391.28} C_VEL
LIN {X 0,Y 509.978,Z 119.77,A -85,B 0,C 180,E1 -5393.67,E2 -5393.67} C_VEL
LIN {X 0,Y 510.055,Z 119.761,A -85,B 0,C 180,E1 -5397.631,E2 -5397.631} C_VEL
LIN {X 0,Y 510.062,Z 119.757,A -85,B 0,C 180,E1 -5400.789,E2 -5400.789} C_VEL
LIN {X 0,Y 509.953,Z 119.772,A -85,B 0,C 180,E1 -5403.16,E2 -5403.16} C_VEL
LIN {X 0,Y 509.977,Z 119.769,A -85,B 0,C 180,E1 -5406.33,E2 -5406.33} C_VEL
LIN {X 0,Y 509.913,Z 119.776,A -85,B 0,C 180,E1 -5408.72,E2 -5408.72} C_VEL
LIN {X 0,Y 509.903,Z 119.78,A -85,B 0,C 180,E1 -5411.932,E2 -5411.932} C_VEL
LIN {X 0,Y 509.892,Z 119.785,A -85,B 0,C 180,E1 -5415.242,E2 -5415.242} C_VEL
LIN {X 0,Y 509.887,Z 119.78,A -85,B 0,C 180,E1 -5418.001,E2 -5418.001} C_VEL
LIN {X 0,Y 509.849,Z 119.79,A -85,B 0,C 180,E1 -5421.002,E2 -5421.002} C_VEL
LIN {X 0,Y 509.862,Z 119.783,A -85,B 0,C 180,E1 -5424.426,E2 -5424.426} C_VEL
LIN {X 0,Y 509.882,Z 119.787,A -85,B 0,C 180,E1 -5427.056,E2 -5427.056} C_VEL
LIN {X 0,Y 509.855,Z 119.783,A -85,B 0,C 180,E1 -5429.751,E2 -5429.751} C_VEL
LIN {X 0,Y 509.871,Z 119.789,A -85,B 0,C 180,E1 -5432.774,E2 -5432.774} C_VEL
LIN {X 0,Y 509.838,Z 119.785,A -85,B 0,C 180,E1 -5435.581,E2 -5435.581} C_VEL
LIN {X 0,Y 509.848,Z 119.79,A -85,B 0,C 180,E1 -5438.338,E2 -5438.338} C_VEL
LIN {X 0,Y 509.855,Z 119.783,A -85,B 0,C 180,E1 -5441.426,E2 -5441.426} C_VEL
LIN {X 0,Y 509.837,Z 119.788,A -85,B 0,C 180,E1 -5444.67,E2 -5444.67} C_VEL
LIN {X 0,Y 509.855,Z 119.791,A -85,B 0,C 180,E1 -5448.103,E2 -5448.103} C_VEL
LIN {X 0,Y 509.844,Z 119.786,A -85,B 0,C 180,E1 -5450.648,E2 -5450.648} C_VEL
LIN {X 0,Y 509.832,Z 119.791,A -85,B 0,C 180,E1 -5453.648,E2 -5453.648} C_VEL
LIN {X 0,Y 509.843,Z 119.785,A -85,B 0,C 180,E1 -5456.538,E2 -5456.538} C_VEL
LIN {X 0,Y 509.844,Z 119.788,A -85,B 0,C 180,E1 -5459.334,E2 -5459.334} C_VEL
LIN {X 0,Y 509.892,Z 119.781,A -85,B 0,C 180,E1 -5462.055,E2 -5462.055} C_VEL
LIN {X 0,Y 509.875,Z 119.782,A -85,B 0,C 180,E1 -5464.704,E2 -5464.704} C_VEL
LIN {X 0,Y 509.899,Z 119.993,A -85,B 0,C 180,E1 -5467.862,E2 -5467.862} C_VEL
LIN {X 0,Y 510.716,Z 125.589,A -85,B 0,C 180,E1 -5469.036,E2 -5469.036} C_VEL
LIN {X 0,Y 510.3,Z 141.135,A -85,B 0,C 180,E1 -5472.106,E2 -5472.106} C_VEL
LIN {X 0,Y 509.94,Z 155.058,A -85,B 0,C 180,E1 -5474.82,E2 -5474.82} C_VEL
LIN {X 0,Y 509.745,Z 169.845,A -85,B 0,C 180,E1 -5477.66,E2 -5477.66} C_VEL
LIN {X 0,Y 509.772,Z 170.84,A -85,B 0,C 180,E1 -5477.752,E2 -5477.752} C_VEL
LIN {X 0,Y 511.049,Z 182.199,A -85,B 0,C 180,E1 -5477.957,E2 -5477.957} C_VEL
LIN {X 0,Y 510.88,Z 246.325,A -85,B 0,C 180,E1 -5478.873,E2 -5478.873} C_VEL
LIN {X 0,Y 510.669,Z 255.503,A -85,B 0,C 180,E1 -5479.092,E2 -5479.092} C_VEL
LIN {X 0,Y 510.548,Z 263.98,A -85,B 0,C 180,E1 -5479.391,E2 -5479.391} C_VEL
LIN {X 0,Y 510.404,Z 272.493,A -85,B 0,C 180,E1 -5479.789,E2 -5479.789} C_VEL
LIN {X 0,Y 510.198,Z 280.837,A -85,B 0,C 180,E1 -5480.285,E2 -5480.285} C_VEL
LIN {X 0,Y 510.018,Z 288.887,A -85,B 0,C 180,E1 -5480.882,E2 -5480.882} C_VEL
LIN {X 0,Y 509.794,Z 296.552,A -85,B 0,C 180,E1 -5481.577,E2 -5481.577} C_VEL
LIN {X 0,Y 509.606,Z 304.592,A -85,B 0,C 180,E1 -5482.472,E2 -5482.472} C_VEL
LIN {X 0,Y 509.447,Z 310.884,A -85,B 0,C 180,E1 -5483.345,E2 -5483.345} C_VEL
LIN {X 0,Y 509.355,Z 317.178,A -85,B 0,C 180,E1 -5484.458,E2 -5484.458} C_VEL
LIN {X 0,Y 509.257,Z 322.354,A -85,B 0,C 180,E1 -5485.647,E2 -5485.647} C_VEL
LIN {X 0,Y 509.245,Z 324.999,A -85,B 0,C 180,E1 -5486.44,E2 -5486.44} C_VEL
LIN {X 0,Y 509.162,Z 327.901,A -85,B 0,C 180,E1 -5487.627,E2 -5487.627} C_VEL
LIN {X 0,Y 509.111,Z 329.152,A -85,B 0,C 180,E1 -5488.418,E2 -5488.418} C_VEL
LIN {X 0,Y 509.071,Z 329.932,A -85,B 0,C 180,E1 -5489.209,E2 -5489.209} C_VEL
LIN {X 0,Y 509.065,Z 330.227,A -85,B 0,C 180,E1 -5490,E2 -5490} C_VEL
LIN {X 0,Y 509.071,Z 329.931,A -85,B 0,C 180,E1 -5490.791,E2 -5490.791} C_VEL
LIN {X 0,Y 509.111,Z 329.151,A -85,B 0,C 180,E1 -5491.582,E2 -5491.582} C_VEL
LIN {X 0,Y 509.162,Z 327.899,A -85,B 0,C 180,E1 -5492.373,E2 -5492.373} C_VEL
LIN {X 0,Y 509.245,Z 324.998,A -85,B 0,C 180,E1 -5493.561,E2 -5493.561} C_VEL
LIN {X 0,Y 509.257,Z 322.352,A -85,B 0,C 180,E1 -5494.353,E2 -5494.353} C_VEL
LIN {X 0,Y 509.355,Z 317.173,A -85,B 0,C 180,E1 -5495.543,E2 -5495.543} C_VEL
LIN {X 0,Y 509.429,Z 310.993,A -85,B 0,C 180,E1 -5496.637,E2 -5496.637} C_VEL
LIN {X 0,Y 509.618,Z 302.889,A -85,B 0,C 180,E1 -5497.728,E2 -5497.728} C_VEL
LIN {X 0,Y 509.804,Z 295.532,A -85,B 0,C 180,E1 -5498.523,E2 -5498.523} C_VEL
LIN {X 0,Y 510.018,Z 287.653,A -85,B 0,C 180,E1 -5499.218,E2 -5499.218} C_VEL
LIN {X 0,Y 510.23,Z 279.329,A -85,B 0,C 180,E1 -5499.814,E2 -5499.814} C_VEL
LIN {X 0,Y 510.465,Z 268.704,A -85,B 0,C 180,E1 -5500.411,E2 -5500.411} C_VEL
LIN {X 0,Y 510.65,Z 257.157,A -85,B 0,C 180,E1 -5500.858,E2 -5500.858} C_VEL
LIN {X 0,Y 510.839,Z 247.511,A -85,B 0,C 180,E1 -5501.105,E2 -5501.105} C_VEL
LIN {X 0,Y 511.035,Z 186.111,A -85,B 0,C 180,E1 -5501.988,E2 -5501.988} C_VEL
LIN {X 0,Y 510.87,Z 179.416,A -85,B 0,C 180,E1 -5502.086,E2 -5502.086} C_VEL
LIN {X 0,Y 509.752,Z 170.403,A -85,B 0,C 180,E1 -5502.269,E2 -5502.269} C_VEL
LIN {X 0,Y 509.953,Z 157.158,A -85,B 0,C 180,E1 -5504.771,E2 -5504.771} C_VEL
LIN {X 0,Y 510.265,Z 142.438,A -85,B 0,C 180,E1 -5507.639,E2 -5507.639} C_VEL
LIN {X 0,Y 510.662,Z 127.248,A -85,B 0,C 180,E1 -5510.634,E2 -5510.634} C_VEL
LIN {X 0,Y 510.513,Z 123.463,A -85,B 0,C 180,E1 -5511.396,E2 -5511.396} C_VEL
LIN {X 0,Y 509.876,Z 119.863,A -85,B 0,C 180,E1 -5512.188,E2 -5512.188} C_VEL
LIN {X 0,Y 509.874,Z 119.782,A -85,B 0,C 180,E1 -5515.296,E2 -5515.296} C_VEL
LIN {X 0,Y 509.897,Z 119.782,A -85,B 0,C 180,E1 -5518.101,E2 -5518.101} C_VEL
LIN {X 0,Y 509.846,Z 119.784,A -85,B 0,C 180,E1 -5521.28,E2 -5521.28} C_VEL
LIN {X 0,Y 509.857,Z 119.791,A -85,B 0,C 180,E1 -5524.203,E2 -5524.203} C_VEL
LIN {X 0,Y 509.817,Z 119.788,A -85,B 0,C 180,E1 -5527.341,E2 -5527.341} C_VEL
LIN {X 0,Y 509.838,Z 119.788,A -85,B 0,C 180,E1 -5530.382,E2 -5530.382} C_VEL
LIN {X 0,Y 509.823,Z 119.787,A -85,B 0,C 180,E1 -5533.062,E2 -5533.062} C_VEL
LIN {X 0,Y 509.823,Z 119.795,A -85,B 0,C 180,E1 -5535.793,E2 -5535.793} C_VEL
LIN {X 0,Y 509.857,Z 119.783,A -85,B 0,C 180,E1 -5538.575,E2 -5538.575} C_VEL
LIN {X 0,Y 509.852,Z 119.788,A -85,B 0,C 180,E1 -5541.787,E2 -5541.787} C_VEL
LIN {X 0,Y 509.844,Z 119.785,A -85,B 0,C 180,E1 -5544.623,E2 -5544.623} C_VEL
LIN {X 0,Y 509.862,Z 119.788,A -85,B 0,C 180,E1 -5547.481,E2 -5547.481} C_VEL
LIN {X 0,Y 509.859,Z 119.782,A -85,B 0,C 180,E1 -5550.274,E2 -5550.274} C_VEL
LIN {X 0,Y 509.885,Z 119.786,A -85,B 0,C 180,E1 -5552.944,E2 -5552.944} C_VEL
LIN {X 0,Y 509.865,Z 119.783,A -85,B 0,C 180,E1 -5555.574,E2 -5555.574} C_VEL
LIN {X 0,Y 509.852,Z 119.79,A -85,B 0,C 180,E1 -5558.998,E2 -5558.998} C_VEL
LIN {X 0,Y 509.89,Z 119.779,A -85,B 0,C 180,E1 -5561.999,E2 -5561.999} C_VEL
LIN {X 0,Y 509.912,Z 119.782,A -85,B 0,C 180,E1 -5564.819,E2 -5564.819} C_VEL
LIN {X 0,Y 509.902,Z 119.78,A -85,B 0,C 180,E1 -5568.124,E2 -5568.124} C_VEL
LIN {X 0,Y 509.916,Z 119.776,A -85,B 0,C 180,E1 -5571.28,E2 -5571.28} C_VEL
LIN {X 0,Y 509.961,Z 119.771,A -85,B 0,C 180,E1 -5573.67,E2 -5573.67} C_VEL
LIN {X 0,Y 510.056,Z 119.76,A -85,B 0,C 180,E1 -5577.631,E2 -5577.631} C_VEL
LIN {X 0,Y 510.065,Z 119.757,A -85,B 0,C 180,E1 -5580.79,E2 -5580.79} C_VEL
LIN {X 0,Y 509.954,Z 119.771,A -85,B 0,C 180,E1 -5583.16,E2 -5583.16} C_VEL
LIN {X 0,Y 509.98,Z 119.77,A -85,B 0,C 180,E1 -5586.33,E2 -5586.33} C_VEL
LIN {X 0,Y 509.916,Z 119.775,A -85,B 0,C 180,E1 -5588.72,E2 -5588.72} C_VEL
LIN {X 0,Y 509.954,Z 119.775,A -85,B 0,C 180,E1 -5591.931,E2 -5591.931} C_VEL
LIN {X 0,Y 509.896,Z 119.783,A -85,B 0,C 180,E1 -5595.242,E2 -5595.242} C_VEL
LIN {X 0,Y 509.884,Z 119.781,A -85,B 0,C 180,E1 -5597.999,E2 -5597.999} C_VEL
LIN {X 0,Y 509.852,Z 119.788,A -85,B 0,C 180,E1 -5601.002,E2 -5601.002} C_VEL
LIN {X 0,Y 509.857,Z 119.783,A -85,B 0,C 180,E1 -5604.427,E2 -5604.427} C_VEL
LIN {X 0,Y 509.886,Z 119.788,A -85,B 0,C 180,E1 -5607.056,E2 -5607.056} C_VEL
LIN {X 0,Y 509.859,Z 119.783,A -85,B 0,C 180,E1 -5609.751,E2 -5609.751} C_VEL
LIN {X 0,Y 509.875,Z 119.788,A -85,B 0,C 180,E1 -5612.774,E2 -5612.774} C_VEL
LIN {X 0,Y 509.841,Z 119.785,A -85,B 0,C 180,E1 -5615.581,E2 -5615.581} C_VEL
LIN {X 0,Y 509.851,Z 119.788,A -85,B 0,C 180,E1 -5618.338,E2 -5618.338} C_VEL
LIN {X 0,Y 509.857,Z 119.783,A -85,B 0,C 180,E1 -5621.426,E2 -5621.426} C_VEL
LIN {X 0,Y 509.84,Z 119.789,A -85,B 0,C 180,E1 -5624.67,E2 -5624.67} C_VEL
LIN {X 0,Y 509.834,Z 119.786,A -85,B 0,C 180,E1 -5627.51,E2 -5627.51} C_VEL
LIN {X 0,Y 509.848,Z 119.786,A -85,B 0,C 180,E1 -5630.648,E2 -5630.648} C_VEL
LIN {X 0,Y 509.832,Z 119.789,A -85,B 0,C 180,E1 -5633.731,E2 -5633.731} C_VEL
LIN {X 0,Y 509.165,Z 119.873,A -85,B 0,C 180,E1 -5634.39,E2 -5634.39} C_VEL
LIN {X 0,Y 506.348,Z 120.222,A -85,B 0,C 180,E1 -5635.462,E2 -5635.462} C_VEL
LIN {X 0,Y 503.956,Z 120.521,A -85,B 0,C 180,E1 -5636.326,E2 -5636.326} C_VEL
LIN {X 0,Y 502.907,Z 120.649,A -85,B 0,C 180,E1 -5636.992,E2 -5636.992} C_VEL
LIN {X 0,Y 502.809,Z 120.661,A -85,B 0,C 180,E1 -5637.217,E2 -5637.217} C_VEL
LIN {X 0,Y 502.817,Z 120.665,A -85,B 0,C 180,E1 -5640.065,E2 -5640.065} C_VEL
LIN {X 0,Y 502.835,Z 120.658,A -85,B 0,C 180,E1 -5642.533,E2 -5642.533} C_VEL
LIN {X 0,Y 502.805,Z 120.665,A -85,B 0,C 180,E1 -5645.305,E2 -5645.305} C_VEL
LIN {X 0,Y 502.782,Z 120.671,A -85,B 0,C 180,E1 -5647.826,E2 -5647.826} C_VEL
LIN {X 0,Y 502.92,Z 120.776,A -85,B 0,C 180,E1 -5650.404,E2 -5650.404} C_VEL
LIN {X 0,Y 503.218,Z 126.497,A -85,B 0,C 180,E1 -5651.75,E2 -5651.75} C_VEL
LIN {X 0,Y 502.884,Z 141.099,A -85,B 0,C 180,E1 -5655.035,E2 -5655.035} C_VEL
LIN {X 0,Y 502.674,Z 152.868,A -85,B 0,C 180,E1 -5657.584,E2 -5657.584} C_VEL
LIN {X 0,Y 502.942,Z 154.895,A -85,B 0,C 180,E1 -5657.671,E2 -5657.671} C_VEL
LIN {X 0,Y 504.198,Z 164.386,A -85,B 0,C 180,E1 -5657.838,E2 -5657.838} C_VEL
LIN {X 0,Y 503.933,Z 228.499,A -85,B 0,C 180,E1 -5658.766,E2 -5658.766} C_VEL
LIN {X 0,Y 503.795,Z 237.663,A -85,B 0,C 180,E1 -5658.992,E2 -5658.992} C_VEL
LIN {X 0,Y 503.678,Z 247.287,A -85,B 0,C 180,E1 -5659.346,E2 -5659.346} C_VEL
LIN {X 0,Y 503.52,Z 255.478,A -85,B 0,C 180,E1 -5659.749,E2 -5659.749} C_VEL
LIN {X 0,Y 503.241,Z 265.093,A -85,B 0,C 180,E1 -5660.352,E2 -5660.352} C_VEL
LIN {X 0,Y 502.995,Z 274.923,A -85,B 0,C 180,E1 -5661.159,E2 -5661.159} C_VEL
LIN {X 0,Y 502.739,Z 282.667,A -85,B 0,C 180,E1 -5661.964,E2 -5661.964} C_VEL
LIN {X 0,Y 502.56,Z 289.033,A -85,B 0,C 180,E1 -5662.769,E2 -5662.769} C_VEL
LIN {X 0,Y 502.523,Z 294.323,A -85,B 0,C 180,E1 -5663.576,E2 -5663.576} C_VEL
LIN {X 0,Y 502.339,Z 298.743,A -85,B 0,C 180,E1 -5664.38,E2 -5664.38} C_VEL
LIN {X 0,Y 502.208,Z 302.425,A -85,B 0,C 180,E1 -5665.183,E2 -5665.183} C_VEL
LIN {X 0,Y 502.264,Z 305.425,A -85,B 0,C 180,E1 -5665.988,E2 -5665.988} C_VEL
LIN {X 0,Y 502.159,Z 307.753,A -85,B 0,C 180,E1 -5666.791,E2 -5666.791} C_VEL
LIN {X 0,Y 502.099,Z 309.529,A -85,B 0,C 180,E1 -5667.593,E2 -5667.593} C_VEL
LIN {X 0,Y 502.036,Z 310.811,A -85,B 0,C 180,E1 -5668.395,E2 -5668.395} C_VEL
LIN {X 0,Y 501.989,Z 311.623,A -85,B 0,C 180,E1 -5669.198,E2 -5669.198} C_VEL
LIN {X 0,Y 501.981,Z 311.932,A -85,B 0,C 180,E1 -5670,E2 -5670} C_VEL
LIN {X 0,Y 501.99,Z 311.659,A -85,B 0,C 180,E1 -5670.802,E2 -5670.802} C_VEL
LIN {X 0,Y 502.037,Z 310.92,A -85,B 0,C 180,E1 -5671.604,E2 -5671.604} C_VEL
LIN {X 0,Y 502.098,Z 309.711,A -85,B 0,C 180,E1 -5672.406,E2 -5672.406} C_VEL
LIN {X 0,Y 502.187,Z 306.865,A -85,B 0,C 180,E1 -5673.61,E2 -5673.61} C_VEL
LIN {X 0,Y 502.276,Z 304.276,A -85,B 0,C 180,E1 -5674.414,E2 -5674.414} C_VEL
LIN {X 0,Y 502.223,Z 301.081,A -85,B 0,C 180,E1 -5675.219,E2 -5675.219} C_VEL
LIN {X 0,Y 502.529,Z 296.022,A -85,B 0,C 180,E1 -5676.222,E2 -5676.222} C_VEL
LIN {X 0,Y 502.529,Z 290.839,A -85,B 0,C 180,E1 -5677.064,E2 -5677.064} C_VEL
LIN {X 0,Y 502.671,Z 285.124,A -85,B 0,C 180,E1 -5677.835,E2 -5677.835} C_VEL
LIN {X 0,Y 502.874,Z 277.866,A -85,B 0,C 180,E1 -5678.641,E2 -5678.641} C_VEL
LIN {X 0,Y 503.143,Z 270.11,A -85,B 0,C 180,E1 -5679.345,E2 -5679.345} C_VEL
LIN {X 0,Y 503.307,Z 261.935,A -85,B 0,C 180,E1 -5679.95,E2 -5679.95} C_VEL
LIN {X 0,Y 503.575,Z 253.403,A -85,B 0,C 180,E1 -5680.453,E2 -5680.453} C_VEL
LIN {X 0,Y 503.739,Z 243.395,A -85,B 0,C 180,E1 -5680.907,E2 -5680.907} C_VEL
LIN {X 0,Y 503.999,Z 231.815,A -85,B 0,C 180,E1 -5681.257,E2 -5681.257} C_VEL
LIN {X 0,Y 503.995,Z 215.039,A -85,B 0,C 180,E1 -5681.534,E2 -5681.534} C_VEL
LIN {X 0,Y 504.084,Z 162.299,A -85,B 0,C 180,E1 -5682.285,E2 -5682.285} C_VEL
LIN {X 0,Y 502.748,Z 153.31,A -85,B 0,C 180,E1 -5682.468,E2 -5682.468} C_VEL
LIN {X 0,Y 502.696,Z 152.218,A -85,B 0,C 180,E1 -5682.618,E2 -5682.618} C_VEL
LIN {X 0,Y 502.952,Z 137.703,A -85,B 0,C 180,E1 -5685.812,E2 -5685.812} C_VEL
LIN {X 0,Y 503.204,Z 126.244,A -85,B 0,C 180,E1 -5688.4,E2 -5688.4} C_VEL
LIN {X 0,Y 502.936,Z 120.757,A -85,B 0,C 180,E1 -5689.701,E2 -5689.701} C_VEL
LIN {X 0,Y 502.789,Z 120.665,A -85,B 0,C 180,E1 -5693.04,E2 -5693.04} C_VEL
LIN {X 0,Y 502.822,Z 120.66,A -85,B 0,C 180,E1 -5695.676,E2 -5695.676} C_VEL
LIN {X 0,Y 502.841,Z 120.665,A -85,B 0,C 180,E1 -5698.372,E2 -5698.372} C_VEL
LIN {X 0,Y 502.793,Z 120.663,A -85,B 0,C 180,E1 -5701.498,E2 -5701.498} C_VEL
LIN {X 0,Y 502.793,Z 120.669,A -85,B 0,C 180,E1 -5703.994,E2 -5703.994} C_VEL
LIN {X 0,Y 502.78,Z 120.665,A -85,B 0,C 180,E1 -5707.178,E2 -5707.178} C_VEL
LIN {X 0,Y 502.787,Z 120.67,A -85,B 0,C 180,E1 -5710.015,E2 -5710.015} C_VEL
LIN {X 0,Y 502.802,Z 120.665,A -85,B 0,C 180,E1 -5712.199,E2 -5712.199} C_VEL
LIN {X 0,Y 502.785,Z 120.669,A -85,B 0,C 180,E1 -5715.47,E2 -5715.47} C_VEL
LIN {X 0,Y 502.819,Z 120.661,A -85,B 0,C 180,E1 -5718.934,E2 -5718.934} C_VEL
LIN {X 0,Y 502.793,Z 120.664,A -85,B 0,C 180,E1 -5722.046,E2 -5722.046} C_VEL
LIN {X 0,Y 502.807,Z 120.666,A -85,B 0,C 180,E1 -5725.035,E2 -5725.035} C_VEL
LIN {X 0,Y 502.782,Z 120.665,A -85,B 0,C 180,E1 -5727.915,E2 -5727.915} C_VEL
LIN {X 0,Y 502.823,Z 120.662,A -85,B 0,C 180,E1 -5730.712,E2 -5730.712} C_VEL
LIN {X 0,Y 502.861,Z 120.657,A -85,B 0,C 180,E1 -5733.439,E2 -5733.439} C_VEL
LIN {X 0,Y 502.784,Z 120.664,A -85,B 0,C 180,E1 -5736.086,E2 -5736.086} C_VEL
LIN {X 0,Y 502.782,Z 120.671,A -85,B 0,C 180,E1 -5738.689,E2 -5738.689} C_VEL
LIN {X 0,Y 502.829,Z 120.66,A -85,B 0,C 180,E1 -5741.248,E2 -5741.248} C_VEL
LIN {X 0,Y 502.821,Z 120.659,A -85,B 0,C 180,E1 -5743.767,E2 -5743.767} C_VEL
LIN {X 0,Y 502.83,Z 120.663,A -85,B 0,C 180,E1 -5746.255,E2 -5746.255} C_VEL
LIN {X 0,Y 502.892,Z 120.655,A -85,B 0,C 180,E1 -5748.717,E2 -5748.717} C_VEL
LIN {X 0,Y 502.9,Z 120.654,A -85,B 0,C 180,E1 -5751.967,E2 -5751.967} C_VEL
LIN {X 0,Y 502.937,Z 120.65,A -85,B 0,C 180,E1 -5754.386,E2 -5754.386} C_VEL
LIN {X 0,Y 503.024,Z 120.636,A -85,B 0,C 180,E1 -5757.598,E2 -5757.598} C_VEL
LIN {X 0,Y 503.026,Z 120.642,A -85,B 0,C 180,E1 -5760,E2 -5760} C_VEL
LIN {X 0,Y 503.024,Z 120.636,A -85,B 0,C 180,E1 -5762.402,E2 -5762.402} C_VEL
LIN {X 0,Y 502.937,Z 120.651,A -85,B 0,C 180,E1 -5765.613,E2 -5765.613} C_VEL
LIN {X 0,Y 502.9,Z 120.653,A -85,B 0,C 180,E1 -5768.033,E2 -5768.033} C_VEL
LIN {X 0,Y 502.876,Z 120.657,A -85,B 0,C 180,E1 -5771.283,E2 -5771.283} C_VEL
LIN {X 0,Y 502.844,Z 120.657,A -85,B 0,C 180,E1 -5774.571,E2 -5774.571} C_VEL
LIN {X 0,Y 502.86,Z 120.656,A -85,B 0,C 180,E1 -5777.907,E2 -5777.907} C_VEL
LIN {X 0,Y 502.827,Z 120.66,A -85,B 0,C 180,E1 -5780.536,E2 -5780.536} C_VEL
LIN {X 0,Y 502.789,Z 120.671,A -85,B 0,C 180,E1 -5783.041,E2 -5783.041} C_VEL
LIN {X 0,Y 502.838,Z 120.658,A -85,B 0,C 180,E1 -5785.676,E2 -5785.676} C_VEL
LIN {X 0,Y 502.838,Z 120.659,A -85,B 0,C 180,E1 -5788.373,E2 -5788.373} C_VEL
LIN {X 0,Y 502.791,Z 120.664,A -85,B 0,C 180,E1 -5791.499,E2 -5791.499} C_VEL
LIN {X 0,Y 502.803,Z 120.667,A -85,B 0,C 180,E1 -5794.444,E2 -5794.444} C_VEL
LIN {X 0,Y 502.779,Z 120.666,A -85,B 0,C 180,E1 -5797.178,E2 -5797.178} C_VEL
LIN {X 0,Y 502.786,Z 120.667,A -85,B 0,C 180,E1 -5800.015,E2 -5800.015} C_VEL
LIN {X 0,Y 502.801,Z 120.668,A -85,B 0,C 180,E1 -5802.199,E2 -5802.199} C_VEL
LIN {X 0,Y 502.783,Z 120.664,A -85,B 0,C 180,E1 -5805.47,E2 -5805.47} C_VEL
LIN {X 0,Y 502.818,Z 120.66,A -85,B 0,C 180,E1 -5808.934,E2 -5808.934} C_VEL
LIN {X 0,Y 502.792,Z 120.671,A -85,B 0,C 180,E1 -5812.046,E2 -5812.046} C_VEL
LIN {X 0,Y 502.803,Z 120.662,A -85,B 0,C 180,E1 -5815.035,E2 -5815.035} C_VEL
LIN {X 0,Y 502.781,Z 120.67,A -85,B 0,C 180,E1 -5817.916,E2 -5817.916} C_VEL
LIN {X 0,Y 502.823,Z 120.659,A -85,B 0,C 180,E1 -5820.712,E2 -5820.712} C_VEL
LIN {X 0,Y 502.862,Z 120.661,A -85,B 0,C 180,E1 -5823.439,E2 -5823.439} C_VEL
LIN {X 0,Y 502.783,Z 120.647,A -85,B 0,C 180,E1 -5826.086,E2 -5826.086} C_VEL
LIN {X 0,Y 502.826,Z 120.719,A -85,B 0,C 180,E1 -5827.677,E2 -5827.677} C_VEL
LIN {X 0,Y 503.647,Z 125.466,A -85,B 0,C 180,E1 -5828.727,E2 -5828.727} C_VEL
LIN {X 0,Y 503.407,Z 138.113,A -85,B 0,C 180,E1 -5831.271,E2 -5831.271} C_VEL
LIN {X 0,Y 502.984,Z 153.886,A -85,B 0,C 180,E1 -5834.397,E2 -5834.397} C_VEL
LIN {X 0,Y 502.7,Z 168.582,A -85,B 0,C 180,E1 -5837.28,E2 -5837.28} C_VEL
LIN {X 0,Y 502.704,Z 170.393,A -85,B 0,C 180,E1 -5837.564,E2 -5837.564} C_VEL
LIN {X 0,Y 504.111,Z 182.962,A -85,B 0,C 180,E1 -5837.801,E2 -5837.801} C_VEL
LIN {X 0,Y 503.936,Z 246.267,A -85,B 0,C 180,E1 -5838.719,E2 -5838.719} C_VEL
LIN {X 0,Y 503.71,Z 255.377,A -85,B 0,C 180,E1 -5838.94,E2 -5838.94} C_VEL
LIN {X 0,Y 503.577,Z 263.854,A -85,B 0,C 180,E1 -5839.242,E2 -5839.242} C_VEL
LIN {X 0,Y 503.41,Z 272.366,A -85,B 0,C 180,E1 -5839.645,E2 -5839.645} C_VEL
LIN {X 0,Y 503.193,Z 280.709,A -85,B 0,C 180,E1 -5840.149,E2 -5840.149} C_VEL
LIN {X 0,Y 502.986,Z 288.758,A -85,B 0,C 180,E1 -5840.754,E2 -5840.754} C_VEL
LIN {X 0,Y 502.74,Z 297.446,A -85,B 0,C 180,E1 -5841.56,E2 -5841.56} C_VEL
LIN {X 0,Y 502.533,Z 305.971,A -85,B 0,C 180,E1 -5842.567,E2 -5842.567} C_VEL
LIN {X 0,Y 502.345,Z 312.658,A -85,B 0,C 180,E1 -5843.574,E2 -5843.574} C_VEL
LIN {X 0,Y 502.282,Z 317.05,A -85,B 0,C 180,E1 -5844.379,E2 -5844.379} C_VEL
LIN {X 0,Y 502.151,Z 322.225,A -85,B 0,C 180,E1 -5845.585,E2 -5845.585} C_VEL
LIN {X 0,Y 502.166,Z 324.871,A -85,B 0,C 180,E1 -5846.389,E2 -5846.389} C_VEL
LIN {X 0,Y 502.067,Z 327.772,A -85,B 0,C 180,E1 -5847.593,E2 -5847.593} C_VEL
LIN {X 0,Y 502.034,Z 329.024,A -85,B 0,C 180,E1 -5848.396,E2 -5848.396} C_VEL
LIN {X 0,Y 501.988,Z 329.804,A -85,B 0,C 180,E1 -5849.198,E2 -5849.198} C_VEL
LIN {X 0,Y 501.98,Z 330.099,A -85,B 0,C 180,E1 -5850,E2 -5850} C_VEL
LIN {X 0,Y 501.988,Z 329.803,A -85,B 0,C 180,E1 -5850.802,E2 -5850.802} C_VEL
LIN {X 0,Y 502.034,Z 329.023,A -85,B 0,C 180,E1 -5851.605,E2 -5851.605} C_VEL
LIN {X 0,Y 502.067,Z 327.771,A -85,B 0,C 180,E1 -5852.407,E2 -5852.407} C_VEL
LIN {X 0,Y 502.166,Z 324.869,A -85,B 0,C 180,E1 -5853.611,E2 -5853.611} C_VEL
LIN {X 0,Y 502.151,Z 322.223,A -85,B 0,C 180,E1 -5854.415,E2 -5854.415} C_VEL
LIN {X 0,Y 502.281,Z 317.045,A -85,B 0,C 180,E1 -5855.621,E2 -5855.621} C_VEL
LIN {X 0,Y 502.366,Z 311.353,A -85,B 0,C 180,E1 -5856.649,E2 -5856.649} C_VEL
LIN {X 0,Y 502.515,Z 304.46,A -85,B 0,C 180,E1 -5857.635,E2 -5857.635} C_VEL
LIN {X 0,Y 502.739,Z 296.425,A -85,B 0,C 180,E1 -5858.542,E2 -5858.542} C_VEL
LIN {X 0,Y 502.986,Z 288.757,A -85,B 0,C 180,E1 -5859.247,E2 -5859.247} C_VEL
LIN {X 0,Y 503.2,Z 280.702,A -85,B 0,C 180,E1 -5859.851,E2 -5859.851} C_VEL
LIN {X 0,Y 503.433,Z 272.359,A -85,B 0,C 180,E1 -5860.355,E2 -5860.355} C_VEL
LIN {X 0,Y 503.567,Z 263.844,A -85,B 0,C 180,E1 -5860.759,E2 -5860.759} C_VEL
LIN {X 0,Y 503.75,Z 253.697,A -85,B 0,C 180,E1 -5861.111,E2 -5861.111} C_VEL
LIN {X 0,Y 503.987,Z 241.29,A -85,B 0,C 180,E1 -5861.37,E2 -5861.37} C_VEL
LIN {X 0,Y 504.035,Z 180.801,A -85,B 0,C 180,E1 -5862.231,E2 -5862.231} C_VEL
LIN {X 0,Y 502.704,Z 170.364,A -85,B 0,C 180,E1 -5862.437,E2 -5862.437} C_VEL
LIN {X 0,Y 502.68,Z 166.48,A -85,B 0,C 180,E1 -5863.132,E2 -5863.132} C_VEL
LIN {X 0,Y 503.024,Z 152.829,A -85,B 0,C 180,E1 -5865.81,E2 -5865.81} C_VEL
LIN {X 0,Y 503.458,Z 137.052,A -85,B 0,C 180,E1 -5868.939,E2 -5868.939} C_VEL
LIN {X 0,Y 503.649,Z 125.456,A -85,B 0,C 180,E1 -5871.273,E2 -5871.273} C_VEL
LIN {X 0,Y 502.827,Z 120.714,A -85,B 0,C 180,E1 -5872.323,E2 -5872.323} C_VEL
LIN {X 0,Y 502.839,Z 120.658,A -85,B 0,C 180,E1 -5875.676,E2 -5875.676} C_VEL
LIN {X 0,Y 502.841,Z 120.665,A -85,B 0,C 180,E1 -5878.373,E2 -5878.373} C_VEL
LIN {X 0,Y 502.793,Z 120.663,A -85,B 0,C 180,E1 -5881.499,E2 -5881.499} C_VEL
LIN {X 0,Y 502.804,Z 120.667,A -85,B 0,C 180,E1 -5883.994,E2 -5883.994} C_VEL
LIN {X 0,Y 502.778,Z 120.665,A -85,B 0,C 180,E1 -5887.178,E2 -5887.178} C_VEL
LIN {X 0,Y 502.788,Z 120.671,A -85,B 0,C 180,E1 -5890.015,E2 -5890.015} C_VEL
LIN {X 0,Y 502.803,Z 120.665,A -85,B 0,C 180,E1 -5892.199,E2 -5892.199} C_VEL
LIN {X 0,Y 502.786,Z 120.668,A -85,B 0,C 180,E1 -5895.47,E2 -5895.47} C_VEL
LIN {X 0,Y 502.821,Z 120.66,A -85,B 0,C 180,E1 -5898.934,E2 -5898.934} C_VEL
LIN {X 0,Y 502.794,Z 120.664,A -85,B 0,C 180,E1 -5902.046,E2 -5902.046} C_VEL
LIN {X 0,Y 502.808,Z 120.665,A -85,B 0,C 180,E1 -5905.035,E2 -5905.035} C_VEL
LIN {X 0,Y 502.784,Z 120.665,A -85,B 0,C 180,E1 -5907.916,E2 -5907.916} C_VEL
LIN {X 0,Y 502.825,Z 120.661,A -85,B 0,C 180,E1 -5910.712,E2 -5910.712} C_VEL
LIN {X 0,Y 502.864,Z 120.657,A -85,B 0,C 180,E1 -5913.439,E2 -5913.439} C_VEL
LIN {X 0,Y 502.786,Z 120.664,A -85,B 0,C 180,E1 -5916.086,E2 -5916.086} C_VEL
LIN {X 0,Y 502.785,Z 120.67,A -85,B 0,C 180,E1 -5918.689,E2 -5918.689} C_VEL
LIN {X 0,Y 502.832,Z 120.66,A -85,B 0,C 180,E1 -5921.248,E2 -5921.248} C_VEL
LIN {X 0,Y 502.823,Z 120.659,A -85,B 0,C 180,E1 -5923.767,E2 -5923.767} C_VEL
LIN {X 0,Y 502.832,Z 120.662,A -85,B 0,C 180,E1 -5926.255,E2 -5926.255} C_VEL
LIN {X 0,Y 502.878,Z 120.657,A -85,B 0,C 180,E1 -5928.717,E2 -5928.717} C_VEL
LIN {X 0,Y 502.903,Z 120.652,A -85,B 0,C 180,E1 -5931.967,E2 -5931.967} C_VEL
LIN {X 0,Y 502.936,Z 120.652,A -85,B 0,C 180,E1 -5934.387,E2 -5934.387} C_VEL
LIN {X 0,Y 503.025,Z 120.635,A -85,B 0,C 180,E1 -5937.598,E2 -5937.598} C_VEL
LIN {X 0,Y 503.029,Z 120.641,A -85,B 0,C 180,E1 -5940,E2 -5940} C_VEL
LIN {X 0,Y 503.026,Z 120.637,A -85,B 0,C 180,E1 -5942.402,E2 -5942.402} C_VEL
LIN {X 0,Y 502.939,Z 120.65,A -85,B 0,C 180,E1 -5945.614,E2 -5945.614} C_VEL
LIN {X 0,Y 502.903,Z 120.654,A -85,B 0,C 180,E1 -5948.033,E2 -5948.033} C_VEL
LIN {X 0,Y 502.895,Z 120.654,A -85,B 0,C 180,E1 -5951.283,E2 -5951.283} C_VEL
LIN {X 0,Y 502.847,Z 120.656,A -85,B 0,C 180,E1 -5954.571,E2 -5954.571} C_VEL
LIN {X 0,Y 502.857,Z 120.657,A -85,B 0,C 180,E1 -5957.907,E2 -5957.907} C_VEL
LIN {X 0,Y 502.831,Z 120.659,A -85,B 0,C 180,E1 -5960.536,E2 -5960.536} C_VEL
LIN {X 0,Y 502.79,Z 120.669,A -85,B 0,C 180,E1 -5963.041,E2 -5963.041} C_VEL
LIN {X 0,Y 502.84,Z 120.659,A -85,B 0,C 180,E1 -5965.676,E2 -5965.676} C_VEL
LIN {X 0,Y 502.842,Z 120.658,A -85,B 0,C 180,E1 -5968.373,E2 -5968.373} C_VEL
LIN {X 0,Y 502.794,Z 120.664,A -85,B 0,C 180,E1 -5971.499,E2 -5971.499} C_VEL
LIN {X 0,Y 502.807,Z 120.665,A -85,B 0,C 180,E1 -5974.444,E2 -5974.444} C_VEL
LIN {X 0,Y 502.782,Z 120.666,A -85,B 0,C 180,E1 -5977.178,E2 -5977.178} C_VEL
LIN {X 0,Y 502.789,Z 120.665,A -85,B 0,C 180,E1 -5980.015,E2 -5980.015} C_VEL
LIN {X 0,Y 502.805,Z 120.666,A -85,B 0,C 180,E1 -5982.199,E2 -5982.199} C_VEL
LIN {X 0,Y 502.787,Z 120.664,A -85,B 0,C 180,E1 -5985.47,E2 -5985.47} C_VEL
LIN {X 0,Y 502.821,Z 120.66,A -85,B 0,C 180,E1 -5988.934,E2 -5988.934} C_VEL
LIN {X 0,Y 502.795,Z 120.67,A -85,B 0,C 180,E1 -5992.046,E2 -5992.046} C_VEL
LIN {X 0,Y 502.806,Z 120.661,A -85,B 0,C 180,E1 -5995.035,E2 -5995.035} C_VEL
LIN {X 0,Y 502.809,Z 120.661,A -85,B 0,C 180,E1 -5997.217,E2 -5997.217} C_VEL
LIN {X 0,Y 502.107,Z 120.757,A -85,B 0,C 180,E1 -5997.886,E2 -5997.886} C_VEL
LIN {X 0,Y 499.243,Z 121.108,A -85,B 0,C 180,E1 -5998.972,E2 -5998.972} C_VEL
LIN {X 0,Y 496.85,Z 121.411,A -85,B 0,C 180,E1 -5999.847,E2 -5999.847} C_VEL
LIN {X 0,Y 495.833,Z 121.531,A -85,B 0,C 180,E1 -6000.522,E2 -6000.522} C_VEL
LIN {X 0,Y 495.755,Z 121.539,A -85,B 0,C 180,E1 -6000.751,E2 -6000.751} C_VEL
LIN {X 0,Y 495.826,Z 121.533,A -85,B 0,C 180,E1 -6003.251,E2 -6003.251} C_VEL
LIN {X 0,Y 495.745,Z 121.543,A -85,B 0,C 180,E1 -6006.612,E2 -6006.612} C_VEL
LIN {X 0,Y 495.841,Z 121.589,A -85,B 0,C 180,E1 -6010.22,E2 -6010.22} C_VEL
LIN {X 0,Y 496.019,Z 122.552,A -85,B 0,C 180,E1 -6010.551,E2 -6010.551} C_VEL
LIN {X 0,Y 496.145,Z 129.946,A -85,B 0,C 180,E1 -6012.269,E2 -6012.269} C_VEL
LIN {X 0,Y 495.838,Z 142.954,A -85,B 0,C 180,E1 -6015.218,E2 -6015.218} C_VEL
LIN {X 0,Y 495.676,Z 153.123,A -85,B 0,C 180,E1 -6017.42,E2 -6017.42} C_VEL
LIN {X 0,Y 495.97,Z 155.47,A -85,B 0,C 180,E1 -6017.501,E2 -6017.501} C_VEL
LIN {X 0,Y 497.285,Z 164.541,A -85,B 0,C 180,E1 -6017.667,E2 -6017.667} C_VEL
LIN {X 0,Y 496.986,Z 228.651,A -85,B 0,C 180,E1 -6018.607,E2 -6018.607} C_VEL
LIN {X 0,Y 496.851,Z 237.807,A -85,B 0,C 180,E1 -6018.836,E2 -6018.836} C_VEL
LIN {X 0,Y 496.709,Z 247.427,A -85,B 0,C 180,E1 -6019.194,E2 -6019.194} C_VEL
LIN {X 0,Y 496.541,Z 255.615,A -85,B 0,C 180,E1 -6019.603,E2 -6019.603} C_VEL
LIN {X 0,Y 496.244,Z 265.228,A -85,B 0,C 180,E1 -6020.215,E2 -6020.215} C_VEL
LIN {X 0,Y 495.973,Z 275.056,A -85,B 0,C 180,E1 -6021.032,E2 -6021.032} C_VEL
LIN {X 0,Y 495.723,Z 282.8,A -85,B 0,C 180,E1 -6021.849,E2 -6021.849} C_VEL
LIN {X 0,Y 495.517,Z 289.165,A -85,B 0,C 180,E1 -6022.666,E2 -6022.666} C_VEL
LIN {X 0,Y 495.455,Z 294.455,A -85,B 0,C 180,E1 -6023.484,E2 -6023.484} C_VEL
LIN {X 0,Y 495.298,Z 298.874,A -85,B 0,C 180,E1 -6024.299,E2 -6024.299} C_VEL
LIN {X 0,Y 495.124,Z 302.555,A -85,B 0,C 180,E1 -6025.114,E2 -6025.114} C_VEL
LIN {X 0,Y 495.185,Z 305.555,A -85,B 0,C 180,E1 -6025.93,E2 -6025.93} C_VEL
LIN {X 0,Y 495.083,Z 307.883,A -85,B 0,C 180,E1 -6026.745,E2 -6026.745} C_VEL
LIN {X 0,Y 495.006,Z 309.658,A -85,B 0,C 180,E1 -6027.559,E2 -6027.559} C_VEL
LIN {X 0,Y 494.962,Z 310.94,A -85,B 0,C 180,E1 -6028.372,E2 -6028.372} C_VEL
LIN {X 0,Y 494.91,Z 311.751,A -85,B 0,C 180,E1 -6029.186,E2 -6029.186} C_VEL
LIN {X 0,Y 494.899,Z 312.06,A -85,B 0,C 180,E1 -6030,E2 -6030} C_VEL
LIN {X 0,Y 494.91,Z 311.787,A -85,B 0,C 180,E1 -6030.813,E2 -6030.813} C_VEL
LIN {X 0,Y 494.963,Z 311.047,A -85,B 0,C 180,E1 -6031.627,E2 -6031.627} C_VEL
LIN {X 0,Y 495.006,Z 309.839,A -85,B 0,C 180,E1 -6032.441,E2 -6032.441} C_VEL
LIN {X 0,Y 495.114,Z 306.992,A -85,B 0,C 180,E1 -6033.662,E2 -6033.662} C_VEL
LIN {X 0,Y 495.184,Z 304.403,A -85,B 0,C 180,E1 -6034.477,E2 -6034.477} C_VEL
LIN {X 0,Y 495.291,Z 299.3,A -85,B 0,C 180,E1 -6035.7,E2 -6035.7} C_VEL
LIN {X 0,Y 495.472,Z 294.979,A -85,B 0,C 180,E1 -6036.515,E2 -6036.515} C_VEL
LIN {X 0,Y 495.496,Z 289.795,A -85,B 0,C 180,E1 -6037.334,E2 -6037.334} C_VEL
LIN {X 0,Y 495.698,Z 283.548,A -85,B 0,C 180,E1 -6038.151,E2 -6038.151} C_VEL
LIN {X 0,Y 495.934,Z 275.952,A -85,B 0,C 180,E1 -6038.968,E2 -6038.968} C_VEL
LIN {X 0,Y 496.194,Z 266.505,A -85,B 0,C 180,E1 -6039.786,E2 -6039.786} C_VEL
LIN {X 0,Y 496.505,Z 257.264,A -85,B 0,C 180,E1 -6040.397,E2 -6040.397} C_VEL
LIN {X 0,Y 496.703,Z 247.138,A -85,B 0,C 180,E1 -6040.909,E2 -6040.909} C_VEL
LIN {X 0,Y 496.917,Z 238.239,A -85,B 0,C 180,E1 -6041.239,E2 -6041.239} C_VEL
LIN {X 0,Y 497.035,Z 228.566,A -85,B 0,C 180,E1 -6041.484,E2 -6041.484} C_VEL
LIN {X 0,Y 497.12,Z 162.487,A -85,B 0,C 180,E1 -6042.458,E2 -6042.458} C_VEL
LIN {X 0,Y 495.689,Z 153.272,A -85,B 0,C 180,E1 -6042.658,E2 -6042.658} C_VEL
LIN {X 0,Y 495.688,Z 150.887,A -85,B 0,C 180,E1 -6043.112,E2 -6043.112} C_VEL
LIN {X 0,Y 495.945,Z 137.764,A -85,B 0,C 180,E1 -6046.041,E2 -6046.041} C_VEL
LIN {X 0,Y 496.201,Z 126.422,A -85,B 0,C 180,E1 -6048.634,E2 -6048.634} C_VEL
LIN {X 0,Y 495.88,Z 121.628,A -85,B 0,C 180,E1 -6049.805,E2 -6049.805} C_VEL
LIN {X 0,Y 495.743,Z 121.541,A -85,B 0,C 180,E1 -6053.387,E2 -6053.387} C_VEL
LIN {X 0,Y 495.824,Z 121.535,A -85,B 0,C 180,E1 -6056.749,E2 -6056.749} C_VEL
LIN {X 0,Y 495.767,Z 121.54,A -85,B 0,C 180,E1 -6059.746,E2 -6059.746} C_VEL
LIN {X 0,Y 495.766,Z 121.541,A -85,B 0,C 180,E1 -6062.594,E2 -6062.594} C_VEL
LIN {X 0,Y 495.754,Z 121.542,A -85,B 0,C 180,E1 -6065.537,E2 -6065.537} C_VEL
LIN {X 0,Y 495.763,Z 121.539,A -85,B 0,C 180,E1 -6068.768,E2 -6068.768} C_VEL
LIN {X 0,Y 495.755,Z 121.547,A -85,B 0,C 180,E1 -6071.781,E2 -6071.781} C_VEL
LIN {X 0,Y 495.736,Z 121.544,A -85,B 0,C 180,E1 -6075.141,E2 -6075.141} C_VEL
LIN {X 0,Y 495.756,Z 121.54,A -85,B 0,C 180,E1 -6078.219,E2 -6078.219} C_VEL
LIN {X 0,Y 495.749,Z 121.548,A -85,B 0,C 180,E1 -6081.408,E2 -6081.408} C_VEL
LIN {X 0,Y 495.755,Z 121.54,A -85,B 0,C 180,E1 -6084.463,E2 -6084.463} C_VEL
LIN {X 0,Y 495.766,Z 121.544,A -85,B 0,C 180,E1 -6087.405,E2 -6087.405} C_VEL
LIN {X 0,Y 495.765,Z 121.538,A -85,B 0,C 180,E1 -6090.253,E2 -6090.253} C_VEL
LIN {X 0,Y 495.822,Z 121.536,A -85,B 0,C 180,E1 -6093.251,E2 -6093.251} C_VEL
LIN {X 0,Y 495.747,Z 121.541,A -85,B 0,C 180,E1 -6095.725,E2 -6095.725} C_VEL
LIN {X 0,Y 495.741,Z 121.544,A -85,B 0,C 180,E1 -6098.371,E2 -6098.371} C_VEL
LIN {X 0,Y 495.784,Z 121.541,A -85,B 0,C 180,E1 -6100.971,E2 -6100.971} C_VEL
LIN {X 0,Y 495.778,Z 121.537,A -85,B 0,C 180,E1 -6103.53,E2 -6103.53} C_VEL
LIN {X 0,Y 495.793,Z 121.537,A -85,B 0,C 180,E1 -6106.056,E2 -6106.056} C_VEL
LIN {X 0,Y 495.867,Z 121.532,A -85,B 0,C 180,E1 -6108.555,E2 -6108.555} C_VEL
LIN {X 0,Y 495.872,Z 121.528,A -85,B 0,C 180,E1 -6111.852,E2 -6111.852} C_VEL
LIN {X 0,Y 495.895,Z 121.529,A -85,B 0,C 180,E1 -6114.306,E2 -6114.306} C_VEL
LIN {X 0,Y 495.993,Z 121.512,A -85,B 0,C 180,E1 -6117.564,E2 -6117.564} C_VEL
LIN {X 0,Y 495.998,Z 121.518,A -85,B 0,C 180,E1 -6120,E2 -6120} C_VEL
LIN {X 0,Y 495.992,Z 121.512,A -85,B 0,C 180,E1 -6122.436,E2 -6122.436} C_VEL
LIN {X 0,Y 495.894,Z 121.53,A -85,B 0,C 180,E1 -6125.693,E2 -6125.693} C_VEL
LIN {X 0,Y 495.871,Z 121.527,A -85,B 0,C 180,E1 -6128.148,E2 -6128.148} C_VEL
LIN {X 0,Y 495.85,Z 121.535,A -85,B 0,C 180,E1 -6131.445,E2 -6131.445} C_VEL
LIN {X 0,Y 495.789,Z 121.537,A -85,B 0,C 180,E1 -6134.783,E2 -6134.783} C_VEL
LIN {X 0,Y 495.786,Z 121.544,A -85,B 0,C 180,E1 -6137.319,E2 -6137.319} C_VEL
LIN {X 0,Y 495.776,Z 121.538,A -85,B 0,C 180,E1 -6139.89,E2 -6139.89} C_VEL
LIN {X 0,Y 495.758,Z 121.544,A -85,B 0,C 180,E1 -6142.861,E2 -6142.861} C_VEL
LIN {X 0,Y 495.788,Z 121.535,A -85,B 0,C 180,E1 -6146.068,E2 -6146.068} C_VEL
LIN {X 0,Y 495.771,Z 121.545,A -85,B 0,C 180,E1 -6148.815,E2 -6148.815} C_VEL
LIN {X 0,Y 495.753,Z 121.54,A -85,B 0,C 180,E1 -6151.725,E2 -6151.725} C_VEL
LIN {X 0,Y 495.773,Z 121.545,A -85,B 0,C 180,E1 -6154.695,E2 -6154.695} C_VEL
LIN {X 0,Y 495.729,Z 121.543,A -85,B 0,C 180,E1 -6157.562,E2 -6157.562} C_VEL
LIN {X 0,Y 495.765,Z 121.543,A -85,B 0,C 180,E1 -6160.7,E2 -6160.7} C_VEL
LIN {X 0,Y 495.727,Z 121.547,A -85,B 0,C 180,E1 -6164.002,E2 -6164.002} C_VEL
LIN {X 0,Y 495.723,Z 121.543,A -85,B 0,C 180,E1 -6167.117,E2 -6167.117} C_VEL
LIN {X 0,Y 495.757,Z 121.546,A -85,B 0,C 180,E1 -6169.953,E2 -6169.953} C_VEL
LIN {X 0,Y 495.728,Z 121.544,A -85,B 0,C 180,E1 -6172.553,E2 -6172.553} C_VEL
LIN {X 0,Y 495.775,Z 121.54,A -85,B 0,C 180,E1 -6175.457,E2 -6175.457} C_VEL
LIN {X 0,Y 495.754,Z 121.541,A -85,B 0,C 180,E1 -6178.364,E2 -6178.364} C_VEL
LIN {X 0,Y 495.787,Z 121.542,A -85,B 0,C 180,E1 -6181.507,E2 -6181.507} C_VEL
LIN {X 0,Y 495.79,Z 121.539,A -85,B 0,C 180,E1 -6183.932,E2 -6183.932} C_VEL
LIN {X 0,Y 495.759,Z 121.518,A -85,B 0,C 180,E1 -6187.14,E2 -6187.14} C_VEL
LIN {X 0,Y 495.802,Z 121.727,A -85,B 0,C 180,E1 -6187.608,E2 -6187.608} C_VEL
LIN {X 0,Y 496.71,Z 128.387,A -85,B 0,C 180,E1 -6189.042,E2 -6189.042} C_VEL
LIN {X 0,Y 496.27,Z 143.252,A -85,B 0,C 180,E1 -6192.061,E2 -6192.061} C_VEL
LIN {X 0,Y 495.867,Z 160.063,A -85,B 0,C 180,E1 -6195.43,E2 -6195.43} C_VEL
LIN {X 0,Y 495.651,Z 170.157,A -85,B 0,C 180,E1 -6197.377,E2 -6197.377} C_VEL
LIN {X 0,Y 497.016,Z 180.873,A -85,B 0,C 180,E1 -6197.596,E2 -6197.596} C_VEL
LIN {X 0,Y 496.989,Z 246.204,A -85,B 0,C 180,E1 -6198.56,E2 -6198.56} C_VEL
LIN {X 0,Y 496.76,Z 255.255,A -85,B 0,C 180,E1 -6198.783,E2 -6198.783} C_VEL
LIN {X 0,Y 496.62,Z 263.73,A -85,B 0,C 180,E1 -6199.09,E2 -6199.09} C_VEL
LIN {X 0,Y 496.423,Z 272.24,A -85,B 0,C 180,E1 -6199.498,E2 -6199.498} C_VEL
LIN {X 0,Y 496.184,Z 280.582,A -85,B 0,C 180,E1 -6200.008,E2 -6200.008} C_VEL
LIN {X 0,Y 495.946,Z 288.631,A -85,B 0,C 180,E1 -6200.621,E2 -6200.621} C_VEL
LIN {X 0,Y 495.7,Z 297.319,A -85,B 0,C 180,E1 -6201.439,E2 -6201.439} C_VEL
LIN {X 0,Y 495.464,Z 305.842,A -85,B 0,C 180,E1 -6202.461,E2 -6202.461} C_VEL
LIN {X 0,Y 495.269,Z 312.53,A -85,B 0,C 180,E1 -6203.482,E2 -6203.482} C_VEL
LIN {X 0,Y 495.211,Z 316.922,A -85,B 0,C 180,E1 -6204.299,E2 -6204.299} C_VEL
LIN {X 0,Y 495.051,Z 322.096,A -85,B 0,C 180,E1 -6205.522,E2 -6205.522} C_VEL
LIN {X 0,Y 495.058,Z 325.897,A -85,B 0,C 180,E1 -6206.745,E2 -6206.745} C_VEL
LIN {X 0,Y 494.976,Z 327.644,A -85,B 0,C 180,E1 -6207.559,E2 -6207.559} C_VEL
LIN {X 0,Y 494.959,Z 328.896,A -85,B 0,C 180,E1 -6208.373,E2 -6208.373} C_VEL
LIN {X 0,Y 494.908,Z 329.676,A -85,B 0,C 180,E1 -6209.187,E2 -6209.187} C_VEL
LIN {X 0,Y 494.897,Z 329.971,A -85,B 0,C 180,E1 -6210,E2 -6210} C_VEL
LIN {X 0,Y 494.908,Z 329.675,A -85,B 0,C 180,E1 -6210.814,E2 -6210.814} C_VEL
LIN {X 0,Y 494.96,Z 328.895,A -85,B 0,C 180,E1 -6211.628,E2 -6211.628} C_VEL
LIN {X 0,Y 494.976,Z 327.642,A -85,B 0,C 180,E1 -6212.441,E2 -6212.441} C_VEL
LIN {X 0,Y 495.088,Z 324.741,A -85,B 0,C 180,E1 -6213.663,E2 -6213.663} C_VEL
LIN {X 0,Y 495.051,Z 322.094,A -85,B 0,C 180,E1 -6214.478,E2 -6214.478} C_VEL
LIN {X 0,Y 495.211,Z 316.916,A -85,B 0,C 180,E1 -6215.702,E2 -6215.702} C_VEL
LIN {X 0,Y 495.336,Z 310.361,A -85,B 0,C 180,E1 -6216.886,E2 -6216.886} C_VEL
LIN {X 0,Y 495.52,Z 302.631,A -85,B 0,C 180,E1 -6217.949,E2 -6217.949} C_VEL
LIN {X 0,Y 495.749,Z 295.273,A -85,B 0,C 180,E1 -6218.766,E2 -6218.766} C_VEL
LIN {X 0,Y 496.008,Z 287.394,A -85,B 0,C 180,E1 -6219.481,E2 -6219.481} C_VEL
LIN {X 0,Y 496.254,Z 279.069,A -85,B 0,C 180,E1 -6220.094,E2 -6220.094} C_VEL
LIN {X 0,Y 496.522,Z 268.442,A -85,B 0,C 180,E1 -6220.707,E2 -6220.707} C_VEL
LIN {X 0,Y 496.733,Z 256.892,A -85,B 0,C 180,E1 -6221.166,E2 -6221.166} C_VEL
LIN {X 0,Y 496.93,Z 247.241,A -85,B 0,C 180,E1 -6221.42,E2 -6221.42} C_VEL
LIN {X 0,Y 497.137,Z 197.492,A -85,B 0,C 180,E1 -6222.16,E2 -6222.16} C_VEL
LIN {X 0,Y 496.977,Z 180.658,A -85,B 0,C 180,E1 -6222.407,E2 -6222.407} C_VEL
LIN {X 0,Y 495.676,Z 170.184,A -85,B 0,C 180,E1 -6222.62,E2 -6222.62} C_VEL
LIN {X 0,Y 495.731,Z 164.255,A -85,B 0,C 180,E1 -6223.737,E2 -6223.737} C_VEL
LIN {X 0,Y 496.126,Z 147.449,A -85,B 0,C 180,E1 -6227.094,E2 -6227.094} C_VEL
LIN {X 0,Y 496.548,Z 133.77,A -85,B 0,C 180,E1 -6229.858,E2 -6229.858} C_VEL
LIN {X 0,Y 496.675,Z 127.156,A -85,B 0,C 180,E1 -6231.211,E2 -6231.211} C_VEL
LIN {X 0,Y 495.803,Z 121.72,A -85,B 0,C 180,E1 -6232.393,E2 -6232.393} C_VEL
LIN {X 0,Y 495.788,Z 121.537,A -85,B 0,C 180,E1 -6235.167,E2 -6235.167} C_VEL
LIN {X 0,Y 495.781,Z 121.538,A -85,B 0,C 180,E1 -6237.891,E2 -6237.891} C_VEL
LIN {X 0,Y 495.752,Z 121.543,A -85,B 0,C 180,E1 -6240.687,E2 -6240.687} C_VEL
LIN {X 0,Y 495.759,Z 121.54,A -85,B 0,C 180,E1 -6243.564,E2 -6243.564} C_VEL
LIN {X 0,Y 495.728,Z 121.545,A -85,B 0,C 180,E1 -6246.544,E2 -6246.544} C_VEL
LIN {X 0,Y 495.757,Z 121.543,A -85,B 0,C 180,E1 -6249.638,E2 -6249.638} C_VEL
LIN {X 0,Y 495.738,Z 121.543,A -85,B 0,C 180,E1 -6252.507,E2 -6252.507} C_VEL
LIN {X 0,Y 495.738,Z 121.543,A -85,B 0,C 180,E1 -6255.141,E2 -6255.141} C_VEL
LIN {X 0,Y 495.757,Z 121.541,A -85,B 0,C 180,E1 -6258.219,E2 -6258.219} C_VEL
LIN {X 0,Y 495.751,Z 121.547,A -85,B 0,C 180,E1 -6261.409,E2 -6261.409} C_VEL
LIN {X 0,Y 495.756,Z 121.539,A -85,B 0,C 180,E1 -6264.463,E2 -6264.463} C_VEL
LIN {X 0,Y 495.768,Z 121.545,A -85,B 0,C 180,E1 -6267.406,E2 -6267.406} C_VEL
LIN {X 0,Y 495.767,Z 121.538,A -85,B 0,C 180,E1 -6270.254,E2 -6270.254} C_VEL
LIN {X 0,Y 495.825,Z 121.537,A -85,B 0,C 180,E1 -6273.251,E2 -6273.251} C_VEL
LIN {X 0,Y 495.748,Z 121.541,A -85,B 0,C 180,E1 -6275.725,E2 -6275.725} C_VEL
LIN {X 0,Y 495.744,Z 121.543,A -85,B 0,C 180,E1 -6278.371,E2 -6278.371} C_VEL
LIN {X 0,Y 495.786,Z 121.541,A -85,B 0,C 180,E1 -6280.972,E2 -6280.972} C_VEL
LIN {X 0,Y 495.781,Z 121.536,A -85,B 0,C 180,E1 -6283.53,E2 -6283.53} C_VEL
LIN {X 0,Y 495.795,Z 121.536,A -85,B 0,C 180,E1 -6286.056,E2 -6286.056} C_VEL
LIN {X 0,Y 495.853,Z 121.535,A -85,B 0,C 180,E1 -6288.555,E2 -6288.555} C_VEL
LIN {X 0,Y 495.874,Z 121.527,A -85,B 0,C 180,E1 -6291.852,E2 -6291.852} C_VEL
LIN {X 0,Y 495.892,Z 121.531,A -85,B 0,C 180,E1 -6294.307,E2 -6294.307} C_VEL
LIN {X 0,Y 495.994,Z 121.511,A -85,B 0,C 180,E1 -6297.564,E2 -6297.564} C_VEL
LIN {X 0,Y 495.985,Z 121.511,A -85,B 0,C 180,E1 -6300.812,E2 -6300.812} C_VEL
LIN {X 0,Y 495.995,Z 121.512,A -85,B 0,C 180,E1 -6302.436,E2 -6302.436} C_VEL
LIN {X 0,Y 495.896,Z 121.528,A -85,B 0,C 180,E1 -6305.694,E2 -6305.694} C_VEL
LIN {X 0,Y 495.875,Z 121.528,A -85,B 0,C 180,E1 -6308.148,E2 -6308.148} C_VEL
LIN {X 0,Y 495.87,Z 121.531,A -85,B 0,C 180,E1 -6311.445,E2 -6311.445} C_VEL
LIN {X 0,Y 495.792,Z 121.535,A -85,B 0,C 180,E1 -6314.783,E2 -6314.783} C_VEL
LIN {X 0,Y 495.784,Z 121.543,A -85,B 0,C 180,E1 -6317.319,E2 -6317.319} C_VEL
LIN {X 0,Y 495.773,Z 121.539,A -85,B 0,C 180,E1 -6319.89,E2 -6319.89} C_VEL
LIN {X 0,Y 495.76,Z 121.542,A -85,B 0,C 180,E1 -6322.86,E2 -6322.86} C_VEL
LIN {X 0,Y 495.791,Z 121.535,A -85,B 0,C 180,E1 -6326.068,E2 -6326.068} C_VEL
LIN {X 0,Y 495.774,Z 121.543,A -85,B 0,C 180,E1 -6328.815,E2 -6328.815} C_VEL
LIN {X 0,Y 495.757,Z 121.539,A -85,B 0,C 180,E1 -6331.725,E2 -6331.725} C_VEL
LIN {X 0,Y 495.777,Z 121.544,A -85,B 0,C 180,E1 -6334.695,E2 -6334.695} C_VEL
LIN {X 0,Y 495.732,Z 121.542,A -85,B 0,C 180,E1 -6337.562,E2 -6337.562} C_VEL
LIN {X 0,Y 495.768,Z 121.544,A -85,B 0,C 180,E1 -6340.7,E2 -6340.7} C_VEL
LIN {X 0,Y 495.729,Z 121.546,A -85,B 0,C 180,E1 -6344.002,E2 -6344.002} C_VEL
LIN {X 0,Y 495.727,Z 121.543,A -85,B 0,C 180,E1 -6347.117,E2 -6347.117} C_VEL
LIN {X 0,Y 495.76,Z 121.544,A -85,B 0,C 180,E1 -6349.953,E2 -6349.953} C_VEL
LIN {X 0,Y 495.732,Z 121.545,A -85,B 0,C 180,E1 -6352.553,E2 -6352.553} C_VEL
LIN {X 0,Y 495.779,Z 121.538,A -85,B 0,C 180,E1 -6355.457,E2 -6355.457} C_VEL
LIN {X 0,Y 495.757,Z 121.542,A -85,B 0,C 180,E1 -6358.364,E2 -6358.364} C_VEL
LIN {X 0,Y 495.755,Z 121.539,A -85,B 0,C 180,E1 -6360.751,E2 -6360.751} C_VEL
LIN {X 0,Y 495.097,Z 121.627,A -85,B 0,C 180,E1 -6361.43,E2 -6361.43} C_VEL
LIN {X 0,Y 492.24,Z 121.978,A -85,B 0,C 180,E1 -6362.533,E2 -6362.533} C_VEL
LIN {X 0,Y 489.827,Z 122.283,A -85,B 0,C 180,E1 -6363.421,E2 -6363.421} C_VEL
LIN {X 0,Y 488.802,Z 122.408,A -85,B 0,C 180,E1 -6364.108,E2 -6364.108} C_VEL
LIN {X 0,Y 488.726,Z 122.415,A -85,B 0,C 180,E1 -6364.34,E2 -6364.34} C_VEL
LIN {X 0,Y 488.724,Z 122.42,A -85,B 0,C 180,E1 -6367.153,E2 -6367.153} C_VEL
LIN {X 0,Y 488.807,Z 122.557,A -85,B 0,C 180,E1 -6370.225,E2 -6370.225} C_VEL
LIN {X 0,Y 489.19,Z 128.139,A -85,B 0,C 180,E1 -6371.575,E2 -6371.575} C_VEL
LIN {X 0,Y 488.856,Z 141.744,A -85,B 0,C 180,E1 -6374.707,E2 -6374.707} C_VEL
LIN {X 0,Y 488.646,Z 153.017,A -85,B 0,C 180,E1 -6377.213,E2 -6377.213} C_VEL
LIN {X 0,Y 488.85,Z 154.914,A -85,B 0,C 180,E1 -6377.306,E2 -6377.306} C_VEL
LIN {X 0,Y 490.35,Z 165.283,A -85,B 0,C 180,E1 -6377.498,E2 -6377.498} C_VEL
LIN {X 0,Y 490.051,Z 228.802,A -85,B 0,C 180,E1 -6378.444,E2 -6378.444} C_VEL
LIN {X 0,Y 489.913,Z 237.949,A -85,B 0,C 180,E1 -6378.676,E2 -6378.676} C_VEL
LIN {X 0,Y 489.746,Z 247.566,A -85,B 0,C 180,E1 -6379.039,E2 -6379.039} C_VEL
LIN {X 0,Y 489.568,Z 255.752,A -85,B 0,C 180,E1 -6379.453,E2 -6379.453} C_VEL
LIN {X 0,Y 489.246,Z 265.363,A -85,B 0,C 180,E1 -6380.074,E2 -6380.074} C_VEL
LIN {X 0,Y 488.971,Z 275.189,A -85,B 0,C 180,E1 -6380.903,E2 -6380.903} C_VEL
LIN {X 0,Y 488.685,Z 282.932,A -85,B 0,C 180,E1 -6381.731,E2 -6381.731} C_VEL
LIN {X 0,Y 488.464,Z 289.297,A -85,B 0,C 180,E1 -6382.56,E2 -6382.56} C_VEL
LIN {X 0,Y 488.378,Z 294.586,A -85,B 0,C 180,E1 -6383.389,E2 -6383.389} C_VEL
LIN {X 0,Y 488.254,Z 299.004,A -85,B 0,C 180,E1 -6384.217,E2 -6384.217} C_VEL
LIN {X 0,Y 488.047,Z 302.685,A -85,B 0,C 180,E1 -6385.043,E2 -6385.043} C_VEL
LIN {X 0,Y 488.092,Z 305.685,A -85,B 0,C 180,E1 -6385.871,E2 -6385.871} C_VEL
LIN {X 0,Y 488.01,Z 308.012,A -85,B 0,C 180,E1 -6386.697,E2 -6386.697} C_VEL
LIN {X 0,Y 487.918,Z 309.788,A -85,B 0,C 180,E1 -6387.523,E2 -6387.523} C_VEL
LIN {X 0,Y 487.891,Z 311.068,A -85,B 0,C 180,E1 -6388.349,E2 -6388.349} C_VEL
LIN {X 0,Y 487.833,Z 311.88,A -85,B 0,C 180,E1 -6389.174,E2 -6389.174} C_VEL
LIN {X 0,Y 487.82,Z 312.188,A -85,B 0,C 180,E1 -6390,E2 -6390} C_VEL
LIN {X 0,Y 487.833,Z 311.915,A -85,B 0,C 180,E1 -6390.825,E2 -6390.825} C_VEL
LIN {X 0,Y 487.891,Z 311.174,A -85,B 0,C 180,E1 -6391.651,E2 -6391.651} C_VEL
LIN {X 0,Y 487.917,Z 309.966,A -85,B 0,C 180,E1 -6392.476,E2 -6392.476} C_VEL
LIN {X 0,Y 488.044,Z 307.119,A -85,B 0,C 180,E1 -6393.715,E2 -6393.715} C_VEL
LIN {X 0,Y 488.098,Z 304.529,A -85,B 0,C 180,E1 -6394.542,E2 -6394.542} C_VEL
LIN {X 0,Y 488.247,Z 299.426,A -85,B 0,C 180,E1 -6395.783,E2 -6395.783} C_VEL
LIN {X 0,Y 488.385,Z 293.946,A -85,B 0,C 180,E1 -6396.816,E2 -6396.816} C_VEL
LIN {X 0,Y 488.544,Z 287.047,A -85,B 0,C 180,E1 -6397.855,E2 -6397.855} C_VEL
LIN {X 0,Y 488.814,Z 279.132,A -85,B 0,C 180,E1 -6398.787,E2 -6398.787} C_VEL
LIN {X 0,Y 489.127,Z 271.583,A -85,B 0,C 180,E1 -6399.511,E2 -6399.511} C_VEL
LIN {X 0,Y 489.313,Z 263.676,A -85,B 0,C 180,E1 -6400.134,E2 -6400.134} C_VEL
LIN {X 0,Y 489.6,Z 255.513,A -85,B 0,C 180,E1 -6400.65,E2 -6400.65} C_VEL
LIN {X 0,Y 489.73,Z 247.256,A -85,B 0,C 180,E1 -6401.066,E2 -6401.066} C_VEL
LIN {X 0,Y 489.981,Z 238.352,A -85,B 0,C 180,E1 -6401.401,E2 -6401.401} C_VEL
LIN {X 0,Y 490.091,Z 228.821,A -85,B 0,C 180,E1 -6401.646,E2 -6401.646} C_VEL
LIN {X 0,Y 490.237,Z 163.458,A -85,B 0,C 180,E1 -6402.623,E2 -6402.623} C_VEL
LIN {X 0,Y 488.693,Z 153.618,A -85,B 0,C 180,E1 -6402.826,E2 -6402.826} C_VEL
LIN {X 0,Y 488.64,Z 152.741,A -85,B 0,C 180,E1 -6402.923,E2 -6402.923} C_VEL
LIN {X 0,Y 488.892,Z 139.702,A -85,B 0,C 180,E1 -6405.85,E2 -6405.85} C_VEL
LIN {X 0,Y 489.187,Z 126.681,A -85,B 0,C 180,E1 -6408.859,E2 -6408.859} C_VEL
LIN {X 0,Y 488.817,Z 122.501,A -85,B 0,C 180,E1 -6409.911,E2 -6409.911} C_VEL
LIN {X 0,Y 488.709,Z 122.419,A -85,B 0,C 180,E1 -6413.02,E2 -6413.02} C_VEL
LIN {X 0,Y 488.728,Z 122.415,A -85,B 0,C 180,E1 -6415.557,E2 -6415.557} C_VEL
LIN {X 0,Y 488.745,Z 122.421,A -85,B 0,C 180,E1 -6418.328,E2 -6418.328} C_VEL
LIN {X 0,Y 488.692,Z 122.419,A -85,B 0,C 180,E1 -6421.179,E2 -6421.179} C_VEL
LIN {X 0,Y 488.728,Z 122.423,A -85,B 0,C 180,E1 -6424.113,E2 -6424.113} C_VEL
LIN {X 0,Y 488.681,Z 122.421,A -85,B 0,C 180,E1 -6427.158,E2 -6427.158} C_VEL
LIN {X 0,Y 488.718,Z 122.419,A -85,B 0,C 180,E1 -6430.344,E2 -6430.344} C_VEL
LIN {X 0,Y 488.684,Z 122.427,A -85,B 0,C 180,E1 -6433.654,E2 -6433.654} C_VEL
LIN {X 0,Y 488.683,Z 122.421,A -85,B 0,C 180,E1 -6436.345,E2 -6436.345} C_VEL
LIN {X 0,Y 488.732,Z 122.42,A -85,B 0,C 180,E1 -6439.676,E2 -6439.676} C_VEL
LIN {X 0,Y 488.681,Z 122.422,A -85,B 0,C 180,E1 -6442.841,E2 -6442.841} C_VEL
LIN {X 0,Y 488.733,Z 122.416,A -85,B 0,C 180,E1 -6445.887,E2 -6445.887} C_VEL
LIN {X 0,Y 488.691,Z 122.423,A -85,B 0,C 180,E1 -6448.82,E2 -6448.82} C_VEL
LIN {X 0,Y 488.743,Z 122.414,A -85,B 0,C 180,E1 -6451.671,E2 -6451.671} C_VEL
LIN {X 0,Y 488.746,Z 122.415,A -85,B 0,C 180,E1 -6454.444,E2 -6454.444} C_VEL
LIN {X 0,Y 488.721,Z 122.42,A -85,B 0,C 180,E1 -6457.153,E2 -6457.153} C_VEL
LIN {X 0,Y 488.728,Z 122.415,A -85,B 0,C 180,E1 -6459.81,E2 -6459.81} C_VEL
LIN {X 0,Y 488.733,Z 122.419,A -85,B 0,C 180,E1 -6462.423,E2 -6462.423} C_VEL
LIN {X 0,Y 488.761,Z 122.413,A -85,B 0,C 180,E1 -6464.999,E2 -6464.999} C_VEL
LIN {X 0,Y 488.829,Z 122.41,A -85,B 0,C 180,E1 -6468.388,E2 -6468.388} C_VEL
LIN {X 0,Y 488.816,Z 122.406,A -85,B 0,C 180,E1 -6471.734,E2 -6471.734} C_VEL
LIN {X 0,Y 488.854,Z 122.407,A -85,B 0,C 180,E1 -6474.224,E2 -6474.224} C_VEL
LIN {X 0,Y 488.96,Z 122.388,A -85,B 0,C 180,E1 -6477.529,E2 -6477.529} C_VEL
LIN {X 0,Y 488.953,Z 122.387,A -85,B 0,C 180,E1 -6480.823,E2 -6480.823} C_VEL
LIN {X 0,Y 488.96,Z 122.387,A -85,B 0,C 180,E1 -6482.471,E2 -6482.471} C_VEL
LIN {X 0,Y 488.854,Z 122.407,A -85,B 0,C 180,E1 -6485.776,E2 -6485.776} C_VEL
LIN {X 0,Y 488.816,Z 122.405,A -85,B 0,C 180,E1 -6488.266,E2 -6488.266} C_VEL
LIN {X 0,Y 488.804,Z 122.413,A -85,B 0,C 180,E1 -6491.612,E2 -6491.612} C_VEL
LIN {X 0,Y 488.761,Z 122.414,A -85,B 0,C 180,E1 -6495,E2 -6495} C_VEL
LIN {X 0,Y 488.753,Z 122.412,A -85,B 0,C 180,E1 -6498.442,E2 -6498.442} C_VEL
LIN {X 0,Y 488.705,Z 122.425,A -85,B 0,C 180,E1 -6501.071,E2 -6501.071} C_VEL
LIN {X 0,Y 488.686,Z 122.421,A -85,B 0,C 180,E1 -6503.746,E2 -6503.746} C_VEL
LIN {X 0,Y 488.79,Z 122.416,A -85,B 0,C 180,E1 -6506.944,E2 -6506.944} C_VEL
LIN {X 0,Y 488.708,Z 122.42,A -85,B 0,C 180,E1 -6510.363,E2 -6510.363} C_VEL
LIN {X 0,Y 488.733,Z 122.415,A -85,B 0,C 180,E1 -6513.484,E2 -6513.484} C_VEL
LIN {X 0,Y 488.686,Z 122.425,A -85,B 0,C 180,E1 -6516.356,E2 -6516.356} C_VEL
LIN {X 0,Y 488.699,Z 122.419,A -85,B 0,C 180,E1 -6519.254,E2 -6519.254} C_VEL
LIN {X 0,Y 488.706,Z 122.418,A -85,B 0,C 180,E1 -6521.6,E2 -6521.6} C_VEL
LIN {X 0,Y 488.699,Z 122.42,A -85,B 0,C 180,E1 -6524.803,E2 -6524.803} C_VEL
LIN {X 0,Y 488.69,Z 122.421,A -85,B 0,C 180,E1 -6527.475,E2 -6527.475} C_VEL
LIN {X 0,Y 488.731,Z 122.418,A -85,B 0,C 180,E1 -6529.677,E2 -6529.677} C_VEL
LIN {X 0,Y 488.68,Z 122.421,A -85,B 0,C 180,E1 -6532.842,E2 -6532.842} C_VEL
LIN {X 0,Y 488.726,Z 122.423,A -85,B 0,C 180,E1 -6535.887,E2 -6535.887} C_VEL
LIN {X 0,Y 488.691,Z 122.42,A -85,B 0,C 180,E1 -6538.82,E2 -6538.82} C_VEL
LIN {X 0,Y 488.744,Z 122.421,A -85,B 0,C 180,E1 -6541.672,E2 -6541.672} C_VEL
LIN {X 0,Y 488.746,Z 122.413,A -85,B 0,C 180,E1 -6544.445,E2 -6544.445} C_VEL
LIN {X 0,Y 488.736,Z 122.497,A -85,B 0,C 180,E1 -6547.433,E2 -6547.433} C_VEL
LIN {X 0,Y 489.727,Z 129.449,A -85,B 0,C 180,E1 -6548.976,E2 -6548.976} C_VEL
LIN {X 0,Y 489.255,Z 144.182,A -85,B 0,C 180,E1 -6552.011,E2 -6552.011} C_VEL
LIN {X 0,Y 488.826,Z 159.938,A -85,B 0,C 180,E1 -6555.215,E2 -6555.215} C_VEL
LIN {X 0,Y 488.603,Z 170.032,A -85,B 0,C 180,E1 -6557.192,E2 -6557.192} C_VEL
LIN {X 0,Y 490.124,Z 181.869,A -85,B 0,C 180,E1 -6557.435,E2 -6557.435} C_VEL
LIN {X 0,Y 490.041,Z 246.134,A -85,B 0,C 180,E1 -6558.397,E2 -6558.397} C_VEL
LIN {X 0,Y 489.798,Z 255.132,A -85,B 0,C 180,E1 -6558.621,E2 -6558.621} C_VEL
LIN {X 0,Y 489.618,Z 264.816,A -85,B 0,C 180,E1 -6558.984,E2 -6558.984} C_VEL
LIN {X 0,Y 489.411,Z 273.991,A -85,B 0,C 180,E1 -6559.45,E2 -6559.45} C_VEL
LIN {X 0,Y 489.087,Z 284.81,A -85,B 0,C 180,E1 -6560.175,E2 -6560.175} C_VEL
LIN {X 0,Y 488.791,Z 293.102,A -85,B 0,C 180,E1 -6560.9,E2 -6560.9} C_VEL
LIN {X 0,Y 488.547,Z 300.8,A -85,B 0,C 180,E1 -6561.729,E2 -6561.729} C_VEL
LIN {X 0,Y 488.376,Z 307.137,A -85,B 0,C 180,E1 -6562.559,E2 -6562.559} C_VEL
LIN {X 0,Y 488.199,Z 312.402,A -85,B 0,C 180,E1 -6563.387,E2 -6563.387} C_VEL
LIN {X 0,Y 488.144,Z 316.794,A -85,B 0,C 180,E1 -6564.216,E2 -6564.216} C_VEL
LIN {X 0,Y 487.959,Z 321.968,A -85,B 0,C 180,E1 -6565.457,E2 -6565.457} C_VEL
LIN {X 0,Y 487.985,Z 325.77,A -85,B 0,C 180,E1 -6566.698,E2 -6566.698} C_VEL
LIN {X 0,Y 487.889,Z 327.516,A -85,B 0,C 180,E1 -6567.523,E2 -6567.523} C_VEL
LIN {X 0,Y 487.887,Z 328.769,A -85,B 0,C 180,E1 -6568.349,E2 -6568.349} C_VEL
LIN {X 0,Y 487.832,Z 329.548,A -85,B 0,C 180,E1 -6569.175,E2 -6569.175} C_VEL
LIN {X 0,Y 487.818,Z 329.843,A -85,B 0,C 180,E1 -6570,E2 -6570} C_VEL
LIN {X 0,Y 487.832,Z 329.547,A -85,B 0,C 180,E1 -6570.826,E2 -6570.826} C_VEL
LIN {X 0,Y 487.887,Z 328.767,A -85,B 0,C 180,E1 -6571.651,E2 -6571.651} C_VEL
LIN {X 0,Y 487.89,Z 327.513,A -85,B 0,C 180,E1 -6572.477,E2 -6572.477} C_VEL
LIN {X 0,Y 488.009,Z 324.612,A -85,B 0,C 180,E1 -6573.716,E2 -6573.716} C_VEL
LIN {X 0,Y 487.959,Z 321.964,A -85,B 0,C 180,E1 -6574.544,E2 -6574.544} C_VEL
LIN {X 0,Y 488.143,Z 316.786,A -85,B 0,C 180,E1 -6575.784,E2 -6575.784} C_VEL
LIN {X 0,Y 488.277,Z 309.962,A -85,B 0,C 180,E1 -6577.028,E2 -6577.028} C_VEL
LIN {X 0,Y 488.463,Z 302.5,A -85,B 0,C 180,E1 -6578.064,E2 -6578.064} C_VEL
LIN {X 0,Y 488.704,Z 295.142,A -85,B 0,C 180,E1 -6578.893,E2 -6578.893} C_VEL
LIN {X 0,Y 489.015,Z 287.263,A -85,B 0,C 180,E1 -6579.618,E2 -6579.618} C_VEL
LIN {X 0,Y 489.256,Z 278.938,A -85,B 0,C 180,E1 -6580.24,E2 -6580.24} C_VEL
LIN {X 0,Y 489.555,Z 268.31,A -85,B 0,C 180,E1 -6580.861,E2 -6580.861} C_VEL
LIN {X 0,Y 489.789,Z 256.757,A -85,B 0,C 180,E1 -6581.327,E2 -6581.327} C_VEL
LIN {X 0,Y 489.977,Z 247.103,A -85,B 0,C 180,E1 -6581.584,E2 -6581.584} C_VEL
LIN {X 0,Y 490.184,Z 203.677,A -85,B 0,C 180,E1 -6582.242,E2 -6582.242} C_VEL
LIN {X 0,Y 490.085,Z 181.65,A -85,B 0,C 180,E1 -6582.568,E2 -6582.568} C_VEL
LIN {X 0,Y 488.616,Z 170.051,A -85,B 0,C 180,E1 -6582.805,E2 -6582.805} C_VEL
LIN {X 0,Y 488.722,Z 163.077,A -85,B 0,C 180,E1 -6584.15,E2 -6584.15} C_VEL
LIN {X 0,Y 489.106,Z 148.375,A -85,B 0,C 180,E1 -6587.132,E2 -6587.132} C_VEL
LIN {X 0,Y 489.588,Z 133.647,A -85,B 0,C 180,E1 -6590.153,E2 -6590.153} C_VEL
LIN {X 0,Y 489.569,Z 127.322,A -85,B 0,C 180,E1 -6591.473,E2 -6591.473} C_VEL
LIN {X 0,Y 488.725,Z 122.494,A -85,B 0,C 180,E1 -6592.568,E2 -6592.568} C_VEL
LIN {X 0,Y 488.747,Z 122.413,A -85,B 0,C 180,E1 -6595.556,E2 -6595.556} C_VEL
LIN {X 0,Y 488.745,Z 122.42,A -85,B 0,C 180,E1 -6598.329,E2 -6598.329} C_VEL
LIN {X 0,Y 488.692,Z 122.419,A -85,B 0,C 180,E1 -6601.18,E2 -6601.18} C_VEL
LIN {X 0,Y 488.731,Z 122.422,A -85,B 0,C 180,E1 -6604.113,E2 -6604.113} C_VEL
LIN {X 0,Y 488.68,Z 122.421,A -85,B 0,C 180,E1 -6607.159,E2 -6607.159} C_VEL
LIN {X 0,Y 488.719,Z 122.419,A -85,B 0,C 180,E1 -6610.345,E2 -6610.345} C_VEL
LIN {X 0,Y 488.684,Z 122.426,A -85,B 0,C 180,E1 -6613.655,E2 -6613.655} C_VEL
LIN {X 0,Y 488.685,Z 122.421,A -85,B 0,C 180,E1 -6616.345,E2 -6616.345} C_VEL
LIN {X 0,Y 488.734,Z 122.421,A -85,B 0,C 180,E1 -6619.677,E2 -6619.677} C_VEL
LIN {X 0,Y 488.682,Z 122.422,A -85,B 0,C 180,E1 -6622.841,E2 -6622.841} C_VEL
LIN {X 0,Y 488.735,Z 122.416,A -85,B 0,C 180,E1 -6625.888,E2 -6625.888} C_VEL
LIN {X 0,Y 488.693,Z 122.422,A -85,B 0,C 180,E1 -6628.82,E2 -6628.82} C_VEL
LIN {X 0,Y 488.745,Z 122.415,A -85,B 0,C 180,E1 -6631.671,E2 -6631.671} C_VEL
LIN {X 0,Y 488.748,Z 122.414,A -85,B 0,C 180,E1 -6634.444,E2 -6634.444} C_VEL
LIN {X 0,Y 488.724,Z 122.421,A -85,B 0,C 180,E1 -6637.153,E2 -6637.153} C_VEL
LIN {X 0,Y 488.726,Z 122.415,A -85,B 0,C 180,E1 -6639.811,E2 -6639.811} C_VEL
LIN {X 0,Y 488.736,Z 122.418,A -85,B 0,C 180,E1 -6642.424,E2 -6642.424} C_VEL
LIN {X 0,Y 488.764,Z 122.414,A -85,B 0,C 180,E1 -6645,E2 -6645} C_VEL
LIN {X 0,Y 488.807,Z 122.412,A -85,B 0,C 180,E1 -6648.388,E2 -6648.388} C_VEL
LIN {X 0,Y 488.819,Z 122.405,A -85,B 0,C 180,E1 -6651.734,E2 -6651.734} C_VEL
LIN {X 0,Y 488.851,Z 122.407,A -85,B 0,C 180,E1 -6654.224,E2 -6654.224} C_VEL
LIN {X 0,Y 488.962,Z 122.387,A -85,B 0,C 180,E1 -6657.529,E2 -6657.529} C_VEL
LIN {X 0,Y 488.936,Z 122.389,A -85,B 0,C 180,E1 -6660.824,E2 -6660.824} C_VEL
LIN {X 0,Y 488.962,Z 122.388,A -85,B 0,C 180,E1 -6662.471,E2 -6662.471} C_VEL
LIN {X 0,Y 488.856,Z 122.406,A -85,B 0,C 180,E1 -6665.776,E2 -6665.776} C_VEL
LIN {X 0,Y 488.819,Z 122.406,A -85,B 0,C 180,E1 -6668.266,E2 -6668.266} C_VEL
LIN {X 0,Y 488.832,Z 122.41,A -85,B 0,C 180,E1 -6671.612,E2 -6671.612} C_VEL
LIN {X 0,Y 488.764,Z 122.412,A -85,B 0,C 180,E1 -6675,E2 -6675} C_VEL
LIN {X 0,Y 488.757,Z 122.411,A -85,B 0,C 180,E1 -6678.442,E2 -6678.442} C_VEL
LIN {X 0,Y 488.708,Z 122.423,A -85,B 0,C 180,E1 -6681.071,E2 -6681.071} C_VEL
LIN {X 0,Y 488.685,Z 122.422,A -85,B 0,C 180,E1 -6683.746,E2 -6683.746} C_VEL
LIN {X 0,Y 488.794,Z 122.413,A -85,B 0,C 180,E1 -6686.944,E2 -6686.944} C_VEL
LIN {X 0,Y 488.711,Z 122.419,A -85,B 0,C 180,E1 -6690.363,E2 -6690.363} C_VEL
LIN {X 0,Y 488.737,Z 122.415,A -85,B 0,C 180,E1 -6693.484,E2 -6693.484} C_VEL
LIN {X 0,Y 488.689,Z 122.423,A -85,B 0,C 180,E1 -6696.355,E2 -6696.355} C_VEL
LIN {X 0,Y 488.702,Z 122.419,A -85,B 0,C 180,E1 -6699.254,E2 -6699.254} C_VEL
LIN {X 0,Y 488.708,Z 122.417,A -85,B 0,C 180,E1 -6701.6,E2 -6701.6} C_VEL
LIN {X 0,Y 488.703,Z 122.421,A -85,B 0,C 180,E1 -6704.803,E2 -6704.803} C_VEL
LIN {X 0,Y 488.693,Z 122.42,A -85,B 0,C 180,E1 -6707.474,E2 -6707.474} C_VEL
LIN {X 0,Y 488.735,Z 122.416,A -85,B 0,C 180,E1 -6709.677,E2 -6709.677} C_VEL
LIN {X 0,Y 488.684,Z 122.421,A -85,B 0,C 180,E1 -6712.841,E2 -6712.841} C_VEL
LIN {X 0,Y 488.729,Z 122.422,A -85,B 0,C 180,E1 -6715.887,E2 -6715.887} C_VEL
LIN {X 0,Y 488.694,Z 122.419,A -85,B 0,C 180,E1 -6718.82,E2 -6718.82} C_VEL
LIN {X 0,Y 488.747,Z 122.42,A -85,B 0,C 180,E1 -6721.671,E2 -6721.671} C_VEL
LIN {X 0,Y 488.726,Z 122.415,A -85,B 0,C 180,E1 -6724.34,E2 -6724.34} C_VEL
LIN {X 0,Y 488.075,Z 122.499,A -85,B 0,C 180,E1 -6725.028,E2 -6725.028} C_VEL
LIN {X 0,Y 485.213,Z 122.859,A -85,B 0,C 180,E1 -6726.145,E2 -6726.145} C_VEL
LIN {X 0,Y 482.778,Z 123.164,A -85,B 0,C 180,E1 -6727.045,E2 -6727.045} C_VEL
LIN {X 0,Y 481.726,Z 123.294,A -85,B 0,C 180,E1 -6727.74,E2 -6727.74} C_VEL
LIN {X 0,Y 481.637,Z 123.303,A -85,B 0,C 180,E1 -6727.976,E2 -6727.976} C_VEL
LIN {X 0,Y 481.785,Z 123.409,A -85,B 0,C 180,E1 -6730.119,E2 -6730.119} C_VEL
LIN {X 0,Y 482.175,Z 128.357,A -85,B 0,C 180,E1 -6731.337,E2 -6731.337} C_VEL
LIN {X 0,Y 481.839,Z 141.633,A -85,B 0,C 180,E1 -6734.434,E2 -6734.434} C_VEL
LIN {X 0,Y 481.587,Z 153.136,A -85,B 0,C 180,E1 -6737.023,E2 -6737.023} C_VEL
LIN {X 0,Y 481.829,Z 154.977,A -85,B 0,C 180,E1 -6737.116,E2 -6737.116} C_VEL
LIN {X 0,Y 483.424,Z 165.58,A -85,B 0,C 180,E1 -6737.318,E2 -6737.318} C_VEL
LIN {X 0,Y 483.104,Z 228.952,A -85,B 0,C 180,E1 -6738.275,E2 -6738.275} C_VEL
LIN {X 0,Y 482.966,Z 238.091,A -85,B 0,C 180,E1 -6738.511,E2 -6738.511} C_VEL
LIN {X 0,Y 482.787,Z 247.704,A -85,B 0,C 180,E1 -6738.879,E2 -6738.879} C_VEL
LIN {X 0,Y 482.6,Z 255.888,A -85,B 0,C 180,E1 -6739.299,E2 -6739.299} C_VEL
LIN {X 0,Y 482.264,Z 265.498,A -85,B 0,C 180,E1 -6739.928,E2 -6739.928} C_VEL
LIN {X 0,Y 481.966,Z 275.322,A -85,B 0,C 180,E1 -6740.77,E2 -6740.77} C_VEL
LIN {X 0,Y 481.647,Z 283.064,A -85,B 0,C 180,E1 -6741.61,E2 -6741.61} C_VEL
LIN {X 0,Y 481.41,Z 289.429,A -85,B 0,C 180,E1 -6742.45,E2 -6742.45} C_VEL
LIN {X 0,Y 481.342,Z 295.533,A -85,B 0,C 180,E1 -6743.439,E2 -6743.439} C_VEL
LIN {X 0,Y 481.209,Z 299.134,A -85,B 0,C 180,E1 -6744.132,E2 -6744.132} C_VEL
LIN {X 0,Y 480.977,Z 302.815,A -85,B 0,C 180,E1 -6744.97,E2 -6744.97} C_VEL
LIN {X 0,Y 481,Z 305.815,A -85,B 0,C 180,E1 -6745.81,E2 -6745.81} C_VEL
LIN {X 0,Y 480.941,Z 308.142,A -85,B 0,C 180,E1 -6746.649,E2 -6746.649} C_VEL
LIN {X 0,Y 480.833,Z 309.917,A -85,B 0,C 180,E1 -6747.487,E2 -6747.487} C_VEL
LIN {X 0,Y 480.793,Z 311.197,A -85,B 0,C 180,E1 -6748.325,E2 -6748.325} C_VEL
LIN {X 0,Y 480.759,Z 312.008,A -85,B 0,C 180,E1 -6749.162,E2 -6749.162} C_VEL
LIN {X 0,Y 480.743,Z 312.316,A -85,B 0,C 180,E1 -6750,E2 -6750} C_VEL
LIN {X 0,Y 480.759,Z 312.043,A -85,B 0,C 180,E1 -6750.837,E2 -6750.837} C_VEL
LIN {X 0,Y 480.793,Z 311.302,A -85,B 0,C 180,E1 -6751.675,E2 -6751.675} C_VEL
LIN {X 0,Y 480.832,Z 310.094,A -85,B 0,C 180,E1 -6752.513,E2 -6752.513} C_VEL
LIN {X 0,Y 480.974,Z 307.246,A -85,B 0,C 180,E1 -6753.77,E2 -6753.77} C_VEL
LIN {X 0,Y 480.998,Z 304.657,A -85,B 0,C 180,E1 -6754.609,E2 -6754.609} C_VEL
LIN {X 0,Y 481.182,Z 299.552,A -85,B 0,C 180,E1 -6755.868,E2 -6755.868} C_VEL
LIN {X 0,Y 481.322,Z 294.547,A -85,B 0,C 180,E1 -6756.831,E2 -6756.831} C_VEL
LIN {X 0,Y 481.511,Z 287.172,A -85,B 0,C 180,E1 -6757.97,E2 -6757.97} C_VEL
LIN {X 0,Y 481.782,Z 279.257,A -85,B 0,C 180,E1 -6758.916,E2 -6758.916} C_VEL
LIN {X 0,Y 482.13,Z 271.706,A -85,B 0,C 180,E1 -6759.65,E2 -6759.65} C_VEL
LIN {X 0,Y 482.323,Z 263.798,A -85,B 0,C 180,E1 -6760.282,E2 -6760.282} C_VEL
LIN {X 0,Y 482.625,Z 255.634,A -85,B 0,C 180,E1 -6760.806,E2 -6760.806} C_VEL
LIN {X 0,Y 482.785,Z 247.374,A -85,B 0,C 180,E1 -6761.227,E2 -6761.227} C_VEL
LIN {X 0,Y 483.02,Z 238.467,A -85,B 0,C 180,E1 -6761.567,E2 -6761.567} C_VEL
LIN {X 0,Y 483.15,Z 229.045,A -85,B 0,C 180,E1 -6761.813,E2 -6761.813} C_VEL
LIN {X 0,Y 483.356,Z 164.474,A -85,B 0,C 180,E1 -6762.793,E2 -6762.793} C_VEL
LIN {X 0,Y 481.647,Z 153.592,A -85,B 0,C 180,E1 -6763.026,E2 -6763.026} C_VEL
LIN {X 0,Y 481.605,Z 152.851,A -85,B 0,C 180,E1 -6763.116,E2 -6763.116} C_VEL
LIN {X 0,Y 481.895,Z 139.778,A -85,B 0,C 180,E1 -6766.087,E2 -6766.087} C_VEL
LIN {X 0,Y 482.173,Z 128.575,A -85,B 0,C 180,E1 -6768.703,E2 -6768.703} C_VEL
LIN {X 0,Y 481.782,Z 123.391,A -85,B 0,C 180,E1 -6769.992,E2 -6769.992} C_VEL
LIN {X 0,Y 481.665,Z 123.295,A -85,B 0,C 180,E1 -6773.201,E2 -6773.201} C_VEL
LIN {X 0,Y 481.69,Z 123.294,A -85,B 0,C 180,E1 -6775.957,E2 -6775.957} C_VEL
LIN {X 0,Y 481.7,Z 123.293,A -85,B 0,C 180,E1 -6778.781,E2 -6778.781} C_VEL
LIN {X 0,Y 481.656,Z 123.304,A -85,B 0,C 180,E1 -6782.189,E2 -6782.189} C_VEL
LIN {X 0,Y 481.688,Z 123.293,A -85,B 0,C 180,E1 -6784.682,E2 -6784.682} C_VEL
LIN {X 0,Y 481.655,Z 123.304,A -85,B 0,C 180,E1 -6788.007,E2 -6788.007} C_VEL
LIN {X 0,Y 481.656,Z 123.296,A -85,B 0,C 180,E1 -6791.041,E2 -6791.041} C_VEL
LIN {X 0,Y 481.654,Z 123.297,A -85,B 0,C 180,E1 -6794.458,E2 -6794.458} C_VEL
LIN {X 0,Y 481.647,Z 123.302,A -85,B 0,C 180,E1 -6797.839,E2 -6797.839} C_VEL
LIN {X 0,Y 481.66,Z 123.296,A -85,B 0,C 180,E1 -6800.654,E2 -6800.654} C_VEL
LIN {X 0,Y 481.63,Z 123.308,A -85,B 0,C 180,E1 -6803.375,E2 -6803.375} C_VEL
LIN {X 0,Y 481.709,Z 123.289,A -85,B 0,C 180,E1 -6806.33,E2 -6806.33} C_VEL
LIN {X 0,Y 481.649,Z 123.301,A -85,B 0,C 180,E1 -6809.417,E2 -6809.417} C_VEL
LIN {X 0,Y 481.699,Z 123.291,A -85,B 0,C 180,E1 -6812.168,E2 -6812.168} C_VEL
LIN {X 0,Y 481.716,Z 123.296,A -85,B 0,C 180,E1 -6814.97,E2 -6814.97} C_VEL
LIN {X 0,Y 481.648,Z 123.297,A -85,B 0,C 180,E1 -6817.705,E2 -6817.705} C_VEL
LIN {X 0,Y 481.707,Z 123.293,A -85,B 0,C 180,E1 -6820.393,E2 -6820.393} C_VEL
LIN {X 0,Y 481.69,Z 123.295,A -85,B 0,C 180,E1 -6823.034,E2 -6823.034} C_VEL
LIN {X 0,Y 481.688,Z 123.292,A -85,B 0,C 180,E1 -6825.639,E2 -6825.639} C_VEL
LIN {X 0,Y 481.794,Z 123.284,A -85,B 0,C 180,E1 -6828.216,E2 -6828.216} C_VEL
LIN {X 0,Y 481.761,Z 123.284,A -85,B 0,C 180,E1 -6831.612,E2 -6831.612} C_VEL
LIN {X 0,Y 481.815,Z 123.284,A -85,B 0,C 180,E1 -6834.139,E2 -6834.139} C_VEL
LIN {X 0,Y 481.927,Z 123.264,A -85,B 0,C 180,E1 -6837.492,E2 -6837.492} C_VEL
LIN {X 0,Y 481.904,Z 123.265,A -85,B 0,C 180,E1 -6840.836,E2 -6840.836} C_VEL
LIN {X 0,Y 481.927,Z 123.263,A -85,B 0,C 180,E1 -6842.507,E2 -6842.507} C_VEL
LIN {X 0,Y 481.815,Z 123.283,A -85,B 0,C 180,E1 -6845.86,E2 -6845.86} C_VEL
LIN {X 0,Y 481.761,Z 123.283,A -85,B 0,C 180,E1 -6848.388,E2 -6848.388} C_VEL
LIN {X 0,Y 481.749,Z 123.289,A -85,B 0,C 180,E1 -6851.785,E2 -6851.785} C_VEL
LIN {X 0,Y 481.741,Z 123.291,A -85,B 0,C 180,E1 -6855.224,E2 -6855.224} C_VEL
LIN {X 0,Y 481.711,Z 123.291,A -85,B 0,C 180,E1 -6858.722,E2 -6858.722} C_VEL
LIN {X 0,Y 481.644,Z 123.302,A -85,B 0,C 180,E1 -6861.395,E2 -6861.395} C_VEL
LIN {X 0,Y 481.672,Z 123.294,A -85,B 0,C 180,E1 -6864.113,E2 -6864.113} C_VEL
LIN {X 0,Y 481.745,Z 123.29,A -85,B 0,C 180,E1 -6867.139,E2 -6867.139} C_VEL
LIN {X 0,Y 481.677,Z 123.293,A -85,B 0,C 180,E1 -6869.741,E2 -6869.741} C_VEL
LIN {X 0,Y 481.67,Z 123.302,A -85,B 0,C 180,E1 -6872.674,E2 -6872.674} C_VEL
LIN {X 0,Y 481.64,Z 123.298,A -85,B 0,C 180,E1 -6875.709,E2 -6875.709} C_VEL
LIN {X 0,Y 481.669,Z 123.298,A -85,B 0,C 180,E1 -6878.859,E2 -6878.859} C_VEL
LIN {X 0,Y 481.651,Z 123.299,A -85,B 0,C 180,E1 -6881.913,E2 -6881.913} C_VEL
LIN {X 0,Y 481.653,Z 123.302,A -85,B 0,C 180,E1 -6884.458,E2 -6884.458} C_VEL
LIN {X 0,Y 481.646,Z 123.301,A -85,B 0,C 180,E1 -6887.839,E2 -6887.839} C_VEL
LIN {X 0,Y 481.678,Z 123.294,A -85,B 0,C 180,E1 -6890.651,E2 -6890.651} C_VEL
LIN {X 0,Y 481.629,Z 123.301,A -85,B 0,C 180,E1 -6893.376,E2 -6893.376} C_VEL
LIN {X 0,Y 481.692,Z 123.293,A -85,B 0,C 180,E1 -6896.329,E2 -6896.329} C_VEL
LIN {X 0,Y 481.649,Z 123.301,A -85,B 0,C 180,E1 -6899.418,E2 -6899.418} C_VEL
LIN {X 0,Y 481.699,Z 123.292,A -85,B 0,C 180,E1 -6902.168,E2 -6902.168} C_VEL
LIN {X 0,Y 481.716,Z 123.286,A -85,B 0,C 180,E1 -6904.97,E2 -6904.97} C_VEL
LIN {X 0,Y 481.718,Z 123.396,A -85,B 0,C 180,E1 -6907.313,E2 -6907.313} C_VEL
LIN {X 0,Y 482.671,Z 129.687,A -85,B 0,C 180,E1 -6908.73,E2 -6908.73} C_VEL
LIN {X 0,Y 482.318,Z 143.009,A -85,B 0,C 180,E1 -6911.523,E2 -6911.523} C_VEL
LIN {X 0,Y 481.823,Z 158.764,A -85,B 0,C 180,E1 -6914.779,E2 -6914.779} C_VEL
LIN {X 0,Y 481.541,Z 169.906,A -85,B 0,C 180,E1 -6917.001,E2 -6917.001} C_VEL
LIN {X 0,Y 482.938,Z 180.457,A -85,B 0,C 180,E1 -6917.226,E2 -6917.226} C_VEL
LIN {X 0,Y 483.346,Z 186.711,A -85,B 0,C 180,E1 -6917.33,E2 -6917.33} C_VEL
LIN {X 0,Y 483.1,Z 246.069,A -85,B 0,C 180,E1 -6918.229,E2 -6918.229} C_VEL
LIN {X 0,Y 482.852,Z 255.011,A -85,B 0,C 180,E1 -6918.455,E2 -6918.455} C_VEL
LIN {X 0,Y 482.66,Z 264.693,A -85,B 0,C 180,E1 -6918.823,E2 -6918.823} C_VEL
LIN {X 0,Y 482.437,Z 273.866,A -85,B 0,C 180,E1 -6919.296,E2 -6919.296} C_VEL
LIN {X 0,Y 482.076,Z 284.684,A -85,B 0,C 180,E1 -6920.031,E2 -6920.031} C_VEL
LIN {X 0,Y 481.71,Z 293.997,A -85,B 0,C 180,E1 -6920.871,E2 -6920.871} C_VEL
LIN {X 0,Y 481.501,Z 300.673,A -85,B 0,C 180,E1 -6921.607,E2 -6921.607} C_VEL
LIN {X 0,Y 481.312,Z 307.01,A -85,B 0,C 180,E1 -6922.449,E2 -6922.449} C_VEL
LIN {X 0,Y 481.106,Z 312.812,A -85,B 0,C 180,E1 -6923.386,E2 -6923.386} C_VEL
LIN {X 0,Y 481.075,Z 316.666,A -85,B 0,C 180,E1 -6924.131,E2 -6924.131} C_VEL
LIN {X 0,Y 480.874,Z 321.84,A -85,B 0,C 180,E1 -6925.39,E2 -6925.39} C_VEL
LIN {X 0,Y 480.914,Z 325.642,A -85,B 0,C 180,E1 -6926.649,E2 -6926.649} C_VEL
LIN {X 0,Y 480.806,Z 327.388,A -85,B 0,C 180,E1 -6927.487,E2 -6927.487} C_VEL
LIN {X 0,Y 480.788,Z 328.64,A -85,B 0,C 180,E1 -6928.325,E2 -6928.325} C_VEL
LIN {X 0,Y 480.758,Z 329.42,A -85,B 0,C 180,E1 -6929.163,E2 -6929.163} C_VEL
LIN {X 0,Y 480.742,Z 329.715,A -85,B 0,C 180,E1 -6930,E2 -6930} C_VEL
LIN {X 0,Y 480.758,Z 329.419,A -85,B 0,C 180,E1 -6930.838,E2 -6930.838} C_VEL
LIN {X 0,Y 480.788,Z 328.638,A -85,B 0,C 180,E1 -6931.675,E2 -6931.675} C_VEL
LIN {X 0,Y 480.806,Z 327.385,A -85,B 0,C 180,E1 -6932.513,E2 -6932.513} C_VEL
LIN {X 0,Y 480.913,Z 324.483,A -85,B 0,C 180,E1 -6933.771,E2 -6933.771} C_VEL
LIN {X 0,Y 480.874,Z 321.835,A -85,B 0,C 180,E1 -6934.611,E2 -6934.611} C_VEL
LIN {X 0,Y 481.072,Z 316.657,A -85,B 0,C 180,E1 -6935.87,E2 -6935.87} C_VEL
LIN {X 0,Y 481.205,Z 309.832,A -85,B 0,C 180,E1 -6937.131,E2 -6937.131} C_VEL
LIN {X 0,Y 481.425,Z 302.37,A -85,B 0,C 180,E1 -6938.183,E2 -6938.183} C_VEL
LIN {X 0,Y 481.69,Z 295.011,A -85,B 0,C 180,E1 -6939.024,E2 -6939.024} C_VEL
LIN {X 0,Y 481.944,Z 288.364,A -85,B 0,C 180,E1 -6939.654,E2 -6939.654} C_VEL
LIN {X 0,Y 482.221,Z 280.309,A -85,B 0,C 180,E1 -6940.285,E2 -6940.285} C_VEL
LIN {X 0,Y 482.454,Z 271.962,A -85,B 0,C 180,E1 -6940.81,E2 -6940.81} C_VEL
LIN {X 0,Y 482.671,Z 263.445,A -85,B 0,C 180,E1 -6941.23,E2 -6941.23} C_VEL
LIN {X 0,Y 482.886,Z 254.126,A -85,B 0,C 180,E1 -6941.571,E2 -6941.571} C_VEL
LIN {X 0,Y 483.163,Z 243.025,A -85,B 0,C 180,E1 -6941.831,E2 -6941.831} C_VEL
LIN {X 0,Y 483.16,Z 182.088,A -85,B 0,C 180,E1 -6942.743,E2 -6942.743} C_VEL
LIN {X 0,Y 481.556,Z 169.968,A -85,B 0,C 180,E1 -6942.993,E2 -6942.993} C_VEL
LIN {X 0,Y 481.655,Z 165.047,A -85,B 0,C 180,E1 -6943.931,E2 -6943.931} C_VEL
LIN {X 0,Y 482.092,Z 149.3,A -85,B 0,C 180,E1 -6947.17,E2 -6947.17} C_VEL
LIN {X 0,Y 482.568,Z 135.629,A -85,B 0,C 180,E1 -6950.014,E2 -6950.014} C_VEL
LIN {X 0,Y 482.55,Z 128.252,A -85,B 0,C 180,E1 -6951.577,E2 -6951.577} C_VEL
LIN {X 0,Y 481.714,Z 123.39,A -85,B 0,C 180,E1 -6952.688,E2 -6952.688} C_VEL
LIN {X 0,Y 481.701,Z 123.293,A -85,B 0,C 180,E1 -6955.957,E2 -6955.957} C_VEL
LIN {X 0,Y 481.7,Z 123.293,A -85,B 0,C 180,E1 -6958.782,E2 -6958.782} C_VEL
LIN {X 0,Y 481.657,Z 123.303,A -85,B 0,C 180,E1 -6962.189,E2 -6962.189} C_VEL
LIN {X 0,Y 481.689,Z 123.294,A -85,B 0,C 180,E1 -6964.682,E2 -6964.682} C_VEL
LIN {X 0,Y 481.655,Z 123.304,A -85,B 0,C 180,E1 -6968.007,E2 -6968.007} C_VEL
LIN {X 0,Y 481.656,Z 123.296,A -85,B 0,C 180,E1 -6971.042,E2 -6971.042} C_VEL
LIN {X 0,Y 481.655,Z 123.297,A -85,B 0,C 180,E1 -6974.458,E2 -6974.458} C_VEL
LIN {X 0,Y 481.648,Z 123.303,A -85,B 0,C 180,E1 -6977.839,E2 -6977.839} C_VEL
LIN {X 0,Y 481.662,Z 123.295,A -85,B 0,C 180,E1 -6980.654,E2 -6980.654} C_VEL
LIN {X 0,Y 481.631,Z 123.306,A -85,B 0,C 180,E1 -6983.376,E2 -6983.376} C_VEL
LIN {X 0,Y 481.711,Z 123.289,A -85,B 0,C 180,E1 -6986.33,E2 -6986.33} C_VEL
LIN {X 0,Y 481.652,Z 123.302,A -85,B 0,C 180,E1 -6989.417,E2 -6989.417} C_VEL
LIN {X 0,Y 481.701,Z 123.29,A -85,B 0,C 180,E1 -6992.168,E2 -6992.168} C_VEL
LIN {X 0,Y 481.718,Z 123.296,A -85,B 0,C 180,E1 -6994.97,E2 -6994.97} C_VEL
LIN {X 0,Y 481.65,Z 123.297,A -85,B 0,C 180,E1 -6997.705,E2 -6997.705} C_VEL
LIN {X 0,Y 481.707,Z 123.292,A -85,B 0,C 180,E1 -7000.393,E2 -7000.393} C_VEL
LIN {X 0,Y 481.693,Z 123.295,A -85,B 0,C 180,E1 -7003.034,E2 -7003.034} C_VEL
LIN {X 0,Y 481.691,Z 123.291,A -85,B 0,C 180,E1 -7005.639,E2 -7005.639} C_VEL
LIN {X 0,Y 481.752,Z 123.288,A -85,B 0,C 180,E1 -7008.215,E2 -7008.215} C_VEL
LIN {X 0,Y 481.764,Z 123.283,A -85,B 0,C 180,E1 -7011.612,E2 -7011.612} C_VEL
LIN {X 0,Y 481.811,Z 123.283,A -85,B 0,C 180,E1 -7014.14,E2 -7014.14} C_VEL
LIN {X 0,Y 481.929,Z 123.263,A -85,B 0,C 180,E1 -7017.493,E2 -7017.493} C_VEL
LIN {X 0,Y 481.888,Z 123.267,A -85,B 0,C 180,E1 -7020.836,E2 -7020.836} C_VEL
LIN {X 0,Y 481.929,Z 123.264,A -85,B 0,C 180,E1 -7022.508,E2 -7022.508} C_VEL
LIN {X 0,Y 481.817,Z 123.284,A -85,B 0,C 180,E1 -7025.86,E2 -7025.86} C_VEL
LIN {X 0,Y 481.764,Z 123.283,A -85,B 0,C 180,E1 -7028.388,E2 -7028.388} C_VEL
LIN {X 0,Y 481.797,Z 123.284,A -85,B 0,C 180,E1 -7031.784,E2 -7031.784} C_VEL
LIN {X 0,Y 481.745,Z 123.289,A -85,B 0,C 180,E1 -7035.224,E2 -7035.224} C_VEL
LIN {X 0,Y 481.714,Z 123.29,A -85,B 0,C 180,E1 -7038.722,E2 -7038.722} C_VEL
LIN {X 0,Y 481.647,Z 123.303,A -85,B 0,C 180,E1 -7041.395,E2 -7041.395} C_VEL
LIN {X 0,Y 481.671,Z 123.294,A -85,B 0,C 180,E1 -7044.114,E2 -7044.114} C_VEL
LIN {X 0,Y 481.748,Z 123.291,A -85,B 0,C 180,E1 -7047.139,E2 -7047.139} C_VEL
LIN {X 0,Y 481.681,Z 123.293,A -85,B 0,C 180,E1 -7049.741,E2 -7049.741} C_VEL
LIN {X 0,Y 481.674,Z 123.3,A -85,B 0,C 180,E1 -7052.674,E2 -7052.674} C_VEL
LIN {X 0,Y 481.643,Z 123.297,A -85,B 0,C 180,E1 -7055.709,E2 -7055.709} C_VEL
LIN {X 0,Y 481.672,Z 123.299,A -85,B 0,C 180,E1 -7058.859,E2 -7058.859} C_VEL
LIN {X 0,Y 481.654,Z 123.298,A -85,B 0,C 180,E1 -7061.913,E2 -7061.913} C_VEL
LIN {X 0,Y 481.656,Z 123.303,A -85,B 0,C 180,E1 -7064.458,E2 -7064.458} C_VEL
LIN {X 0,Y 481.649,Z 123.299,A -85,B 0,C 180,E1 -7067.839,E2 -7067.839} C_VEL
LIN {X 0,Y 481.682,Z 123.295,A -85,B 0,C 180,E1 -7070.651,E2 -7070.651} C_VEL
LIN {X 0,Y 481.632,Z 123.3,A -85,B 0,C 180,E1 -7073.376,E2 -7073.376} C_VEL
LIN {X 0,Y 481.695,Z 123.294,A -85,B 0,C 180,E1 -7076.329,E2 -7076.329} C_VEL
LIN {X 0,Y 481.652,Z 123.299,A -85,B 0,C 180,E1 -7079.417,E2 -7079.417} C_VEL
LIN {X 0,Y 481.702,Z 123.293,A -85,B 0,C 180,E1 -7082.168,E2 -7082.168} C_VEL
LIN {X 0,Y 481.695,Z 123.292,A -85,B 0,C 180,E1 -7084.969,E2 -7084.969} C_VEL
LIN {X 0,Y 481.637,Z 123.303,A -85,B 0,C 180,E1 -7087.976,E2 -7087.976} C_VEL
LIN {X 0,Y 480.954,Z 123.39,A -85,B 0,C 180,E1 -7088.452,E2 -7088.452} C_VEL
LIN {X 0,Y 475.443,Z 124.441,A -85,B 0,C 180,E1 -7089.935,E2 -7089.935} C_VEL
LIN {X 0,Y 474.933,Z 125.674,A -85,B 0,C 180,E1 -7090.378,E2 -7090.378} C_VEL
LIN {X 0,Y 475.179,Z 130.456,A -85,B 0,C 180,E1 -7091.544,E2 -7091.544} C_VEL
LIN {X 0,Y 474.819,Z 143.218,A -85,B 0,C 180,E1 -7094.548,E2 -7094.548} C_VEL
LIN {X 0,Y 474.576,Z 153.351,A -85,B 0,C 180,E1 -7096.837,E2 -7096.837} C_VEL
LIN {X 0,Y 474.802,Z 154.961,A -85,B 0,C 180,E1 -7096.919,E2 -7096.919} C_VEL
LIN {X 0,Y 476.484,Z 165.742,A -85,B 0,C 180,E1 -7097.13,E2 -7097.13} C_VEL
LIN {X 0,Y 476.17,Z 229.101,A -85,B 0,C 180,E1 -7098.102,E2 -7098.102} C_VEL
LIN {X 0,Y 476.025,Z 238.233,A -85,B 0,C 180,E1 -7098.341,E2 -7098.341} C_VEL
LIN {X 0,Y 475.825,Z 247.842,A -85,B 0,C 180,E1 -7098.714,E2 -7098.714} C_VEL
LIN {X 0,Y 475.617,Z 257.893,A -85,B 0,C 180,E1 -7099.248,E2 -7099.248} C_VEL
LIN {X 0,Y 475.192,Z 268.324,A -85,B 0,C 180,E1 -7099.992,E2 -7099.992} C_VEL
LIN {X 0,Y 474.909,Z 276.474,A -85,B 0,C 180,E1 -7100.739,E2 -7100.739} C_VEL
LIN {X 0,Y 474.633,Z 283.196,A -85,B 0,C 180,E1 -7101.485,E2 -7101.485} C_VEL
LIN {X 0,Y 474.363,Z 289.56,A -85,B 0,C 180,E1 -7102.337,E2 -7102.337} C_VEL
LIN {X 0,Y 474.261,Z 294.848,A -85,B 0,C 180,E1 -7103.191,E2 -7103.191} C_VEL
LIN {X 0,Y 474.141,Z 299.265,A -85,B 0,C 180,E1 -7104.044,E2 -7104.044} C_VEL
LIN {X 0,Y 473.912,Z 302.945,A -85,B 0,C 180,E1 -7104.895,E2 -7104.895} C_VEL
LIN {X 0,Y 473.916,Z 307.124,A -85,B 0,C 180,E1 -7106.173,E2 -7106.173} C_VEL
LIN {X 0,Y 473.752,Z 310.046,A -85,B 0,C 180,E1 -7107.449,E2 -7107.449} C_VEL
LIN {X 0,Y 473.698,Z 311.326,A -85,B 0,C 180,E1 -7108.299,E2 -7108.299} C_VEL
LIN {X 0,Y 473.687,Z 312.136,A -85,B 0,C 180,E1 -7109.15,E2 -7109.15} C_VEL
LIN {X 0,Y 473.67,Z 312.444,A -85,B 0,C 180,E1 -7110,E2 -7110} C_VEL
LIN {X 0,Y 473.688,Z 312.171,A -85,B 0,C 180,E1 -7110.85,E2 -7110.85} C_VEL
LIN {X 0,Y 473.699,Z 311.43,A -85,B 0,C 180,E1 -7111.7,E2 -7111.7} C_VEL
LIN {X 0,Y 473.751,Z 310.221,A -85,B 0,C 180,E1 -7112.551,E2 -7112.551} C_VEL
LIN {X 0,Y 473.905,Z 307.372,A -85,B 0,C 180,E1 -7113.826,E2 -7113.826} C_VEL
LIN {X 0,Y 473.902,Z 304.784,A -85,B 0,C 180,E1 -7114.678,E2 -7114.678} C_VEL
LIN {X 0,Y 474.121,Z 299.679,A -85,B 0,C 180,E1 -7115.956,E2 -7115.956} C_VEL
LIN {X 0,Y 474.276,Z 293.235,A -85,B 0,C 180,E1 -7117.193,E2 -7117.193} C_VEL
LIN {X 0,Y 474.553,Z 285.622,A -85,B 0,C 180,E1 -7118.302,E2 -7118.302} C_VEL
LIN {X 0,Y 474.808,Z 278.362,A -85,B 0,C 180,E1 -7119.156,E2 -7119.156} C_VEL
LIN {X 0,Y 475.13,Z 271.829,A -85,B 0,C 180,E1 -7119.794,E2 -7119.794} C_VEL
LIN {X 0,Y 475.34,Z 263.92,A -85,B 0,C 180,E1 -7120.435,E2 -7120.435} C_VEL
LIN {X 0,Y 475.662,Z 255.754,A -85,B 0,C 180,E1 -7120.966,E2 -7120.966} C_VEL
LIN {X 0,Y 475.831,Z 247.492,A -85,B 0,C 180,E1 -7121.393,E2 -7121.393} C_VEL
LIN {X 0,Y 476.075,Z 238.581,A -85,B 0,C 180,E1 -7121.738,E2 -7121.738} C_VEL
LIN {X 0,Y 476.219,Z 229.29,A -85,B 0,C 180,E1 -7121.985,E2 -7121.985} C_VEL
LIN {X 0,Y 476.411,Z 164.926,A -85,B 0,C 180,E1 -7122.977,E2 -7122.977} C_VEL
